(* CODESYS project Prepare.project

Project tree, tasks and I/O mapping:
  Device : CODESYS Control x86 Arca Control SM, 3S - Smart Software Solutions GmbH, version 3.5.8.0
    application Application
      libraries: Standard, * (System); Network, 3.5.7.0 (3S - Smart Software Solutions GmbH); Arca Motion Library, 1.0.4.14 (BonMET)
      task MainTask (cyclic, interval t#20ms, priority 1) calls Main
      hand blocks/
        function block AuxAxis_PowerOn [ST]
        data type Grab_Command
        function block Grab_Control [ST]
        function block Grab_Demo [ST]
        data type Grab_State
        function block Hand_Gesture [ST]
        data type Gesture_Type
        data type Error_Message
        function block Hand_Gesture_Demo [ST]
      program Main [ST]
      function block Organize_Hand_Command [ST]
      CNC Execute/
        function block CNC_Execute_Manager [ST]
      simple_functions/
        function block Value_Clamp [ST]
      TCPIP Control/
        data type Robot_Command_via_tcp
        data type Robot_State
        function block TCP_Command_Extract_And_Analysis [ST]
        function block TCPServerConnection [ST]
      Vision Control/
        function block Vision_Control [ST]
      global variables GVL
    SoftMotion General Axis Pool
*)

// Device/Application/hand blocks/Grab_Command
TYPE Grab_Command :
STRUCT
	Tip_Angle : REAL;
	Root_Angle : REAL;
	Clamp_Angle : REAL;
END_STRUCT
END_TYPE

// Device/Application/hand blocks/Grab_State
TYPE Grab_State :
STRUCT
	Tip_State : BOOL;
	Root_State : BOOL;
	Clamp_Angle : REAL;
END_STRUCT
END_TYPE

// Device/Application/hand blocks/Gesture_Type
{attribute 'qualified_only'}
{attribute 'strict'}
TYPE Gesture_Type :
(
	Gesture_Type_None			:= 0,
	Gesture_Type_Num_1		:= 1,
	Gesture_Type_Num_2		:= 2,
	Gesture_Type_Num_3		:= 3,
	Gesture_Type_Num_4		:= 4,
	Gesture_Type_Num_5		:= 5,
	Gesture_Type_Num_6		:= 6,
	Gesture_Type_Fist			:= 10,
	Gesture_Type_Palm			:= 11,
	Gesture_Type_ThumbUp		:= 12,
	Gesture_Type_ThumbDown	:= 13,
	Gesture_Type_ComeOnBaby	:= 14,
	Gesture_Type_PointTo		:= 15,
	Gesture_Type_Wave			:= 16,
	Gesture_Type_Nya			:= 17,
	Gesture_Type_MovObj			:= 18
);
END_TYPE

// Device/Application/hand blocks/Error_Message
{attribute 'qualified_only'}
{attribute 'strict'}
TYPE Error_Message :
(
	Err_None := 0,
	
	Err_AuxAxis_Movement_Cannot_read_virture_robot_position := 10,	// gesture block not reading robot position
	Err_Gesture_Type_Hand_Pos_Not_Given := 20,	// gesture block not given position
	Err_AuxAxis_Movement_Block_err := 30,	// gesture block first reset movement block err
	Err_Gesture_Type_Cycle_mov_block_err := 40,	// gesture block cycle movement block err
	
	Err_PowerOn_Block_Err := 50,
	Err_PowerOn_TimeOut := 51,
	
	Err_Power_Reset_Block_Err := 60,
	Err_Power_Reset_TimeOut := 61,
	
	Err_Group_Enable_Block_Err := 70,
	Err_Group_Enable_TimeOut := 71
);
END_TYPE

// Device/Application/TCPIP Control/Robot_Command_via_tcp
TYPE Robot_Command_via_tcp :
STRUCT
	X_Axis_Valid : BOOL;
	X_value : REAL;
	Y_Axis_Valid : BOOL;
	Y_value : REAL;
	Z_Axis_Valid : BOOL;
	Z_value : REAL;
	Spin : BOOL;
	Grab_Valid : BOOL;
	Grab_state : BOOL := FALSE;
	Gesture_Valid : BOOL;
	Gesture_Num : Gesture_Type;
	Enabl_Hand_Valid : BOOL;
	Enabl_Hand_state : BOOL;
	Gesture_Demo_Valid : BOOL;
	Gesture_Demo_state : BOOL;
	CNC_Mov_Valid : BOOL;
	CNC_Mov_Program_Num : INT;
END_STRUCT
END_TYPE

// Device/Application/TCPIP Control/Robot_State
TYPE Robot_State :
STRUCT
	Hand_Enabled : BOOL;
	Hand_Enb_Err : BOOL;
	Grab_State : BOOL;
	Gesture_State : Gesture_Type := gesture_type.Gesture_Type_None;
	Hand_Mov_Err : BOOL;
	Robot_Mov_Err : BOOL;
	CNC_Executing : BOOL;
	CNC_Execute_Done : BOOL;
	CNC_Execute_Err : BOOL;
END_STRUCT
END_TYPE

// Device/Application/GVL
VAR_GLOBAL
	AllAxisGroupEnb : BOOL := FALSE;
END_VAR

// Device/Application/Main
PROGRAM Main
VAR
	// manual function
	enable_internal : BOOL;
	MoveEn:BOOL:=FALSE;
	enb_triger : r_trig;
	disenb_triger : r_trig;
	
	start_hand_demo_internal : BOOL;
	demo_triger : r_trig;
	
	GestInternal: BOOL;
	GestTypeInternal:INT;
	Gest_triger : R_TRIG;
	
	// auto function
	TCP_Server : TCPserverconnection;
	commandOut : TCP_Command_Extract_And_Analysis;
	handMov : Organize_Hand_Command;
	Execute_CNC_Via_TCP : CNC_Execute_Manager;
	vision : vision_control;
	hand_cmd_valid : BOOL;
	hand_cmd : robot_command_via_tcp;
	old_pos_ready, new_pos_ready : BOOL;
	pick_triger, release_triger : R_TRIG;
	
	//debug
	ToqueT : ARRAY [0..13] OF ArcaLibrary.MCAT_AxisSetLimits;
	Texe : BOOL;
	Tdone, Terr : ARRAY [0..13] OF BOOL;
	SpL, TqL : ARRAY [1..13] OF REAL;
	ToqueState : INT := 0;
	axisOffset : INT := 13;
	axisMaxNum : INT := 25;
	i : INT;
	debug_auto_torque : BOOL;
	ToqueLimit: REAL := 0.5;
	
	AxisM : ARRAY [1..13] OF MCAT_ReadAxisMeasures;
	Aenb : BOOL := TRUE;
	Availd : ARRAY [1..13] OF BOOL;
	AtqM : ARRAY [1..13] OF REAL;
	
	tryRPow : ARRAY [1..13] OF ArcaLibrary.MCAT_ReadPowerStatus;
	PowS : ARRAY [1..13] OF byte;
	clk: INT;
	
	
	/// one button on
	EnableOld:BOOL:=FALSE;
	Status:INT;
	GoToZero:BOOL:=FALSE;
	CycleDone:BOOL;
	
	MoveAbsBlocks:ARRAY[0..5] OF ArcaLibrary.MC_MoveAbsolute;
	PosZero : ARRAY[0..5] OF REAL := [0.0,  18.0, 32.0, 0.0, 0.0, 0.0];
	ExecuteZero:BOOL:=FALSE;
	SpeedZero:REAL:=0.1;
	AccelZero:REAL:=5.0;
	DecelZero:REAL:=5.0;
	JerkZero:REAL:=50.0;
	ZeroError:BOOL;
	ZeroDone:BOOL;
	
	AxPos:ARRAY[1..12] OF REAL;
	AxPosRef:ARRAY[1..12] OF REAL;
	AxReadMea:ARRAY[1..12] OF ArcaLibrary.MCAT_ReadAxisMeasures;
	AxReadRef:ARRAY[1..12] OF ArcaLibrary.MCAT_ReadAxisRef;
	
	AxMoveAbs : ArcaLibrary.MC_MoveAbsolute;
	AxMoveAbs2 : ArcaLibrary.MC_MoveAbsolute;
	AxMoveEn:BOOL:=FALSE;
	AxMoveN:INT:=0;
	AxMovePos:REAL:=0;
	AxMoveVel:REAL:=1;
	AxMoveAcc:REAL:=1;
	AxMoveJerk:REAL:=25.0;
	AxMoveDone:BOOL;
	AxMoveDone2:BOOL;
	
	GrpEn:ArcaLibrary.MC_GroupEnable;
	GrpDis:ArcaLibrary.MC_GroupDisable;
	GrpEnDone, GrpEnErr:BOOL;
	GrpRead:ArcaLibrary.MC_GroupReadActualPosition;
	GrpPos:ARRAY[1..6] OF REAL;

	//initial position of the tool:
	Pos1 : ARRAY[0..5] OF REAL := [0.36, 0.000, 0.7, 0.000, 10, -180.000];
	Pos2 : ARRAY[0..5] OF REAL := [0.36, 0.010, 0.65, 0.000, 10, -180.000];
	Pos3 : ARRAY[0..5] OF REAL := [0.36, -0.010, 0.7, 0.000, 10, -180.000];
	Pos4 : ARRAY[0..5] OF REAL := [0.36, 0.000, 0.65, 0.000, 10, -180.000];
	
	Posleft : ARRAY[0..5] OF REAL := [-60.0,  7.0, 27.0, 0.0, 0.0, 0.0];
	Posright : ARRAY[0..5] OF REAL := [-50.0,  9.0, 30.0, 0.0, 0.0, 0.0];
	
	
	ToolMoveAbs1, ToolMoveAbs2, ToolMoveAbs3, ToolMoveAbs4, ToolMoveAbs5, ToolMoveAbs6 : ArcaLibrary.MC_MoveLinearAbsolute;
	ToolMoveDone1, ToolMoveDone2, ToolMoveDone3, ToolMoveDone4, ToolMoveDone5, ToolMoveDone6 :BOOL;
	
	ToolMoveVel:REAL:=1;
	ToolMoveAcc:REAL:=100;
	ToolMoveJrk:REAL:=1000;
	
	BlendMov : ArcaLibrary.MC_BUFFER_MODE := mcBuffered;
	TransMov : ArcaLibrary.MC_TRANSITION_MODE := tmCornerDistance;	
	TransPar : REAL := 0.0;
	
	ReadDI: ArcaLibrary.BMET_Read_DI;
	ReadDO: ArcaLibrary.BMET_Read_DO;
	WriteDO: ArcaLibrary.BMET_Write_DO;
	ValueRead : UINT;
	ValueDO : UINT;
	LampActivate : UINT;
	
	J : INT := 0;
	DelayTimer : Ton;
END_VAR

//	manually operation process
enb_triger (clk := enable_internal);
disenb_triger (clk := NOT enable_internal);
demo_triger (clk := start_hand_demo_internal);
Gest_triger (clk := GestInternal);

//*****************
TCP_Server(enable := TRUE, outDataReady := commandout.Response_Valid,
	 OutData := commandout.Response ,outDataSize := commandout.Response_Data_Size);

commandout(indata := tcp_server.InData 
	, inDataSize := TCP_Server.InDataSize
	, inData_Valid := TCP_Server.InDataReady
	, OutRobot_State := handmov.Current_Hand_State
	);
	
hand_cmd_valid := commandout.Command_Valid OR pick_triger.Q OR release_triger.Q OR enb_triger.Q
	OR disenb_triger.Q OR demo_triger.Q
	OR Gest_triger.Q;
hand_cmd := commandout.Command;
IF pick_triger.Q THEN
	hand_cmd.Gesture_Valid := TRUE;
	hand_cmd.Gesture_Num := 10;
END_IF
IF release_triger.Q THEN
	hand_cmd.Gesture_Valid := TRUE;
	hand_cmd.Gesture_Num := 11;
END_IF
IF enb_triger.Q THEN
	hand_cmd.Enabl_Hand_Valid := TRUE;
	hand_cmd.Enabl_Hand_state := TRUE;
END_IF
IF disenb_triger.Q THEN
	hand_cmd.Enabl_Hand_Valid := TRUE;
	hand_cmd.Enabl_Hand_state := FALSE;
END_IF
IF demo_triger.Q THEN
	hand_cmd.Gesture_Demo_Valid := TRUE;
	hand_cmd.Gesture_Demo_state := TRUE;
END_IF
IF Gest_triger.Q THEN
	hand_cmd.Gesture_Valid := TRUE;
	hand_cmd.Gesture_Num := GestTypeInternal;
END_IF

handMov(enable:= TRUE, new_cmd_valid := hand_cmd_valid
	, new_cmd := hand_cmd
	);

Execute_CNC_Via_TCP(enable := TRUE, mov_group := 1
	, Tcp_cmd_valid := commandout.Command_Valid
	, TCP_CMD := commandout.Command
	);
(*	dont where has conflict, after enable second robot keep sotping cannot move
vision(enable := handmov.Current_Hand_State.Hand_Enabled, robot_group := 1
	, execute := vision.ready
	, wait_signal_before_pick := TRUE, isPicked := handmov.Current_Hand_State.Gesture_State = 10
	, delay_release_obj := T#2S
	);

pick_triger(clk := vision.ready_to_pick);
release_triger(clk := vision.ready_to_release);
*)
(*************************
	Toque test above
**************************)
ToqueT[01](Execute := Texe, Axis := 06, SpeedLimit := SpL[01], TorqueLimit := TqL[01], Done => Tdone[01], Error => Terr [01]);
ToqueT[02](Execute := Texe, Axis := 07, SpeedLimit := SpL[02], TorqueLimit := TqL[02], Done => Tdone[02], Error => Terr [02]);
ToqueT[03](Execute := Texe, Axis := 08, SpeedLimit := SpL[03], TorqueLimit := TqL[03], Done => Tdone[03], Error => Terr [03]);
ToqueT[04](Execute := Texe, Axis := 09, SpeedLimit := SpL[04], TorqueLimit := TqL[04], Done => Tdone[04], Error => Terr [04]);
ToqueT[05](Execute := Texe, Axis := 10, SpeedLimit := SpL[05], TorqueLimit := TqL[05], Done => Tdone[05], Error => Terr [05]);
ToqueT[06](Execute := Texe, Axis := 11, SpeedLimit := SpL[06], TorqueLimit := TqL[06], Done => Tdone[06], Error => Terr [06]);
ToqueT[07](Execute := Texe, Axis := 12, SpeedLimit := SpL[07], TorqueLimit := TqL[07], Done => Tdone[07], Error => Terr [07]);
ToqueT[08](Execute := Texe, Axis := 13, SpeedLimit := SpL[08], TorqueLimit := TqL[08], Done => Tdone[08], Error => Terr [08]);
ToqueT[09](Execute := Texe, Axis := 14, SpeedLimit := SpL[09], TorqueLimit := TqL[09], Done => Tdone[09], Error => Terr [09]);
ToqueT[10](Execute := Texe, Axis := 15, SpeedLimit := SpL[10], TorqueLimit := TqL[10], Done => Tdone[10], Error => Terr [10]);
ToqueT[11](Execute := Texe, Axis := 16, SpeedLimit := SpL[11], TorqueLimit := TqL[11], Done => Tdone[11], Error => Terr [11]);

// auto set toque limit after axis enabled
CASE ToqueState OF 
	0:
		IF handMov.Current_Hand_State.Hand_Enabled AND NOT debug_auto_torque THEN
			i := 0;
			toquestate := 10;
		END_IF
	10:
		ToqueT[i](Execute := TRUE, Axis := axisOffset + i, TorqueLimit := ToqueLimit, Done => Tdone[i], Error => Terr [i]);
		IF Tdone[i] THEN
			i := i + 1;
			IF axisOffset + i > axisMaxNum THEN
				i := 0;
				toquestate := 20;
			END_IF
		END_IF
	20:
		ToqueT[i](Execute := FALSE);
		i := i + 1;
		IF axisOffset + i > axisMaxNum THEN
			toquestate := 30;
		END_IF
	30:
		IF NOT handMov.Current_Hand_State.Hand_Enabled THEN
			toquestate := 0;
		END_IF
END_CASE

AxisM[01](enable := Aenb, Axis := 6, Torque=> AtqM[01]);
AxisM[02](enable := Aenb, Axis := 7, Torque=> AtqM[02]);
AxisM[03](enable := Aenb, Axis := 8, Torque=> AtqM[03]);
AxisM[04](enable := Aenb, Axis := 9, Torque=> AtqM[04]);
AxisM[05](enable := Aenb, Axis := 10, Torque=> AtqM[05]);
AxisM[06](enable := Aenb, Axis := 11, Torque=> AtqM[06]);
AxisM[07](enable := Aenb, Axis := 12, Torque=> AtqM[07]);
AxisM[08](enable := Aenb, Axis := 13, Torque=> AtqM[08]);
AxisM[09](enable := Aenb, Axis := 14, Torque=> AtqM[09]);
AxisM[10](enable := Aenb, Axis := 15, Torque=> AtqM[10]);
AxisM[11](enable := Aenb, Axis := 16, Torque=> AtqM[11]);

tryRPow[01](enable := TRUE, axis := 06, state=> pows[01]);
tryRPow[02](enable := TRUE, axis := 07, state=> pows[01]);
tryRPow[03](enable := TRUE, axis := 08, state=> pows[01]);
tryRPow[04](enable := TRUE, axis := 09, state=> pows[01]);
tryRPow[05](enable := TRUE, axis := 10, state=> pows[01]);
tryRPow[06](enable := TRUE, axis := 11, state=> pows[01]);
tryRPow[07](enable := TRUE, axis := 12, state=> pows[01]);
tryRPow[08](enable := TRUE, axis := 13, state=> pows[01]);
tryRPow[09](enable := TRUE, axis := 14, state=> pows[01]);
tryRPow[10](enable := TRUE, axis := 15, state=> pows[01]);
tryRPow[11](enable := TRUE, axis := 16, state=> pows[01]);


(***********************
one button start mov
************************)
// read of  measures
AxReadMea[1](Axis:=0, Enable:=(Status>=3 AND Status<100), Pos=>AxPos[1]);
AxReadMea[2](Axis:=1, Enable:=(Status>=3 AND Status<100), Pos=>AxPos[2]);
AxReadMea[3](Axis:=2, Enable:=(Status>=3 AND Status<100), Pos=>AxPos[3]);
AxReadMea[4](Axis:=3, Enable:=(Status>=3 AND Status<100), Pos=>AxPos[4]);
AxReadMea[5](Axis:=4, Enable:=(Status>=3 AND Status<100), Pos=>AxPos[5]);
AxReadMea[6](Axis:=5, Enable:=(Status>=3 AND Status<100), Pos=>AxPos[6]);
AxReadMea[7](Axis:=6, Enable:=(Status>=3 AND Status<100), Pos=>AxPos[7]);
AxReadMea[8](Axis:=7, Enable:=(Status>=3 AND Status<100), Pos=>AxPos[8]);
AxReadMea[9](Axis:=8, Enable:=(Status>=3 AND Status<100), Pos=>AxPos[9]);
AxReadMea[10](Axis:=9, Enable:=(Status>=3 AND Status<100), Pos=>AxPos[10]);
AxReadMea[11](Axis:=10, Enable:=(Status>=3 AND Status<100), Pos=>AxPos[11]);
AxReadMea[12](Axis:=11, Enable:=(Status>=3 AND Status<100), Pos=>AxPos[12]);
// read of reference
AxReadRef[1](Axis:=0, Enable:=(Status>=3 AND Status<100), PosRef=>AxPosRef[1]);
AxReadRef[2](Axis:=1, Enable:=(Status>=3 AND Status<100), PosRef=>AxPosRef[2]);
AxReadRef[3](Axis:=2, Enable:=(Status>=3 AND Status<100), PosRef=>AxPosRef[3]);
AxReadRef[4](Axis:=3, Enable:=(Status>=3 AND Status<100), PosRef=>AxPosRef[4]);
AxReadRef[5](Axis:=4, Enable:=(Status>=3 AND Status<100), PosRef=>AxPosRef[5]);
AxReadRef[6](Axis:=5, Enable:=(Status>=3 AND Status<100), PosRef=>AxPosRef[6]);
AxReadRef[7](Axis:=6, Enable:=(Status>=3 AND Status<100), PosRef=>AxPosRef[7]);
AxReadRef[8](Axis:=7, Enable:=(Status>=3 AND Status<100), PosRef=>AxPosRef[8]);
AxReadRef[9](Axis:=8, Enable:=(Status>=3 AND Status<100), PosRef=>AxPosRef[9]);
AxReadRef[10](Axis:=9, Enable:=(Status>=3 AND Status<100), PosRef=>AxPosRef[10]);
AxReadRef[11](Axis:=10, Enable:=(Status>=3 AND Status<100), PosRef=>AxPosRef[11]);
AxReadRef[12](Axis:=11, Enable:=(Status>=3 AND Status<100), PosRef=>AxPosRef[12]);
// read group position MCS
GrpRead(AxesGroup:=0, Execute:=(Status>=3 AND Status<100), 
	CoordSystem:=ArcaLibrary.MC_COORD_SYSTEM.mcMcs, Position=>GrpPos);

// Powered acquisition from panel 读轴的输入输出
ReadDI(Axis:=0,Enable:=TRUE,Value=>ValueRead);
ReadDO(Axis:=0,Enable:=TRUE,Value=>ValueDO);
WriteDO(Axis:=0,Enable:=TRUE,Value:=0, Mask:=15);


//Press EnableServo to turn on the motors
IF (ValueRead=8) THEN
	J := J + 1;
	IF (J>50) THEN
		enable_internal:=TRUE;
	END_IF
END_IF
//if Button EnableServo is pressed for more than 1 second, turn off the motors
IF (ValueRead=8 AND J > 150) THEN  //OR (ValueRead=0) THEN
	enable_internal:=FALSE;
	MoveEn:=FALSE;
	J:=0;
END_IF

//
// State machines
//
IF (NOT enable_internal) THEN
	WriteDO(Axis:=0,Enable:=TRUE,Value:=0,Mask:=15);
	Status:=0;
ELSE
	WriteDO(Axis:=0,Enable:=TRUE,Value:=2,Mask:=15);
END_IF

//ReadDigitalInput as MoveEnable
IF (ValueRead=16) THEN
	MoveEn:=TRUE;
END_IF
IF (ValueRead=32) THEN
	MoveEn:=FALSE;
END_IF

CASE (Status) OF
	
	//// OFF
	0:
	IF (enable_internal) THEN
		WriteDO(Axis:=0,Enable:=TRUE,Value:=2,Mask:=15);
		Status:=1;
	END_IF
	
	//// POWERING ON
	1:
		IF AllAxisGroupEnb THEN
			Status:=2;
		END_IF
	
	//// IDLE - WAIT FOR COMMAND
	2:
		IF moveEn THEN
			AxMoveAbs(Axis:=11, execute := FALSE);
			status := 3;
		END_IF
	// FORWARD KINEMATIC
	3:
		WriteDO(Axis:=0,Enable:=TRUE,Value:=3,Mask:=15);
		IF NOT moveEn THEN
			status := 2;
		END_IF
			
		// move 5axis of robot 1, in order to move robot later
		AxMoveAbs(Axis:=11, Execute:=TRUE, Position:=80, Velocity:=10, 
			Acceleration:=10, Deceleration:=10, Jerk:=10, 
			BufferMode:=ArcaLibrary.MC_BUFFER_MODE.mcAborting, Done=>AxMoveDone);
					
		IF AxMoveDone THEN
			AxMoveAbs(Axis:=11, execute := FALSE);
			status := 4;
		END_IF
	
	// GROUP MOVEMENT - START
	4:
		WriteDO(Axis:=0,Enable:=TRUE,Value:=6,Mask:=15);
		IF (NOT MoveEn) THEN
			WriteDO(Axis:=0,Enable:=TRUE,Value:=3,Mask:=15);
			Status:=3;
		END_IF
		
		CycleDone:=FALSE;
		// clear block status
		ToolMoveAbs1(AxesGroup:=1, Execute:=FALSE);
		ToolMoveAbs2(AxesGroup:=1, Execute:=FALSE);
		ToolMoveAbs3(AxesGroup:=1, Execute:=FALSE);
		ToolMoveAbs4(AxesGroup:=1, Execute:=FALSE);
		ToolMoveAbs5(AxesGroup:=1, Execute:=FALSE);
		ToolMoveAbs6(AxesGroup:=1, Execute:=FALSE);
		Status:=5;
		DelayTimer(in:= FALSE);
		CycleDone:=FALSE;
		GestInternal := FALSE;
		
			
	// GROUP MOVEMENT - FIRST MOVEMENT
	5:
		WriteDO(Axis:=0,Enable:=TRUE,Value:=6,Mask:=15);
		IF (NOT MoveEn) THEN
			Status:=3;
		END_IF
		
		IF (NOT CycleDone) THEN
			ToolMoveAbs1(AxesGroup:=1, Execute:=TRUE, Position:=ADR(Pos1), Velocity:=ToolMoveVel, Acceleration:=ToolMoveAcc,
				Deceleration:=ToolMoveAcc, Jerk:=ToolMoveJrk, CoordSystem:=mcMcs 
				, TransitionMode := tmNone
				, BufferMode:=mcBuffered, Done=>ToolMoveDone1);
		END_IF
		
		IF (ToolMoveDone1) THEN
			GestInternal := TRUE;
			GestTypeInternal := 1;
			DelayTimer(in:= TRUE, pt := T#5000MS);
			IF delaytimer.Q THEN
				DelayTimer(in:= FALSE);
				GestInternal := FALSE;
				Status:= 51;
				ToolMoveDone1 := FALSE;
			END_IF
		END_IF
	
		
	// GROUP MOVEMENT - SECOND MOVEMENT
	51:
		WriteDO(Axis:=0,Enable:=TRUE,Value:=6,Mask:=15);
		IF (NOT MoveEn) THEN
			Status:=3;
		END_IF
		
		IF (NOT CycleDone) THEN
			ToolMoveAbs2(AxesGroup:=1, Execute:=TRUE, Position:=ADR(Pos2), Velocity:=ToolMoveVel, Acceleration:=ToolMoveAcc,
				Deceleration:=ToolMoveAcc, Jerk:=ToolMoveJrk, CoordSystem:=ArcaLibrary.MC_COORD_SYSTEM.mcMcs, 
				BufferMode:=BlendMov, TransitionMode:=TransMov, TransitionParameter:=ADR(TransPar), Done=>ToolMoveDone2);
		END_IF
		
		IF (ToolMoveDone2) THEN
			GestInternal := TRUE;
			GestTypeInternal := 2;
			DelayTimer(in:= TRUE, pt := T#5000MS);
			IF delaytimer.Q THEN
				DelayTimer(in:= FALSE);
				GestInternal := FALSE;
				Status:=52;
			END_IF
		END_IF

	// GROUP MOVEMENT - THIRD MOVEMENT
	52:
		WriteDO(Axis:=0,Enable:=TRUE,Value:=6,Mask:=15);
		IF (NOT MoveEn) THEN
			Status:=3;
		END_IF
		
		IF (NOT CycleDone) THEN
			ToolMoveAbs3(AxesGroup:=1, Execute:=TRUE, Position:=ADR(Pos3), Velocity:=ToolMoveVel, Acceleration:=ToolMoveAcc,
				Deceleration:=ToolMoveAcc, Jerk:=ToolMoveJrk, CoordSystem:=ArcaLibrary.MC_COORD_SYSTEM.mcMcs, 
				BufferMode:=BlendMov, TransitionMode:=TransMov, TransitionParameter:=ADR(TransPar), Done=>ToolMoveDone3);
		END_IF
		
		IF (ToolMoveDone3) THEN
			GestInternal := TRUE;
			GestTypeInternal := 3;
			DelayTimer(in:= TRUE, pt := T#5000MS);
			IF delaytimer.Q THEN
				DelayTimer(in:= FALSE);
				GestInternal := FALSE;
				Status:=4;
			END_IF
		END_IF

	// GROUP MOVEMENT - FOURTH MOVEMENT
	53:
		WriteDO(Axis:=0,Enable:=TRUE,Value:=6,Mask:=15);
		IF (NOT MoveEn) THEN
			Status:=3;
		END_IF
		
		IF (NOT CycleDone) THEN
			ToolMoveAbs4(AxesGroup:=1, Execute:=TRUE, Position:=ADR(Pos4), Velocity:=ToolMoveVel, Acceleration:=ToolMoveAcc,
				Deceleration:=ToolMoveAcc, Jerk:=ToolMoveJrk, CoordSystem:=ArcaLibrary.MC_COORD_SYSTEM.mcMcs, 
				BufferMode:=mcBuffered, Done=>ToolMoveDone4);
		END_IF

		IF (ToolMoveDone4) THEN
			Status:=4;
		END_IF

	// GROUP MOVEMENT - FIFTH MOVEMENT
	54:
		WriteDO(Axis:=0,Enable:=TRUE,Value:=6,Mask:=15);
		IF (NOT MoveEn) THEN
			Status:=3;
		END_IF
		
		IF (NOT CycleDone) THEN
	//		ToolMoveAbs5(AxesGroup:=1, Execute:=TRUE, Position:=ADR(Pos4), Velocity:=ToolMoveVel, Acceleration:=ToolMoveAcc,
	//			Deceleration:=ToolMoveAcc, Jerk:=ToolMoveJrk, CoordSystem:=ArcaLibrary.MC_COORD_SYSTEM.mcMcs, 
	//			BufferMode:=BlendMov, TransitionMode:=TransMov, TransitionParameter:=ADR(TransPar), Done=>ToolMoveDone5);
		END_IF

		IF (ToolMoveDone5) THEN
			Status:=55;
		END_IF

	// GROUP MOVEMENT - SIXTH MOVEMENT
	55:
		WriteDO(Axis:=0,Enable:=TRUE,Value:=6,Mask:=15);
		IF (NOT MoveEn) THEN
			Status:=3;
		END_IF
		
		IF (NOT CycleDone) THEN
	//		ToolMoveAbs6(AxesGroup:=1, Execute:=TRUE, Position:=ADR(Pos3), Velocity:=ToolMoveVel, Acceleration:=ToolMoveAcc,
	//			Deceleration:=ToolMoveAcc, Jerk:=ToolMoveJrk, CoordSystem:=ArcaLibrary.MC_COORD_SYSTEM.mcMcs, 
	//			BufferMode:=BlendMov, TransitionMode:=TransMov, TransitionParameter:=ADR(TransPar), Done=>ToolMoveDone6);
		END_IF

		IF (ToolMoveDone6) THEN
			CycleDone:=TRUE;
			Status:=4;
		END_IF


	//// ERROR
	100:
		WriteDO(Axis:=0,Enable:=TRUE,Value:=3,Mask:=15);
	
	
END_CASE

END_PROGRAM

// Device/Application/TCPIP Control/TCPServerConnection
FUNCTION_BLOCK TCPServerConnection
VAR_INPUT
	Enable : BOOL;
	OutDataReady : BOOL;
	OutDataSize : CAA.SIZE;
	OutData :  ARRAY [0..255] OF BYTE;;
END_VAR
VAR_OUTPUT
	Err : BOOL;
	InDataReady : BOOL;
	InDataSize : CAA.SIZE;
	InData : STRING;
END_VAR
VAR
	TCPServer : NBS.TCP_Server;
	IP_Addr : NBS.IP_ADDR := (sAddr :='192.168.80.240');
	Port: UINT := 23; // TCP/IP port
	TCPS_Err : BOOL := FALSE;
	TCPS_Err_Mssage : NBS.ERROR;
	
	TCPS_Connection : NBS.TCP_Connection;
	
	ServerRead : NBS.TCP_Read;
	ServerSend : NBS.TCP_Write;
	
	Hendle_enable :BOOL;
	Some_Connect_In : BOOL;
	
	// message out
	_OutDataSize : CAA.SIZE;
	debug : BOOL;
	testTXT :STRING := '0123456';
	testByte : ARRAY [0..5] OF BYTE := [40,12,41,40,10,41];
	ddone, deErr, dxErr : BOOL;
END_VAR

// initialize TCP server
TCPServer(xEnable := Enable, ipAddr := IP_Addr, uiPort := Port, xError => TCPS_Err, eError => TCPS_Err_Mssage);

// send handle after there are some client connect 
TCPS_Connection(xEnable := Hendle_enable, hServer := TCPServer.hServer);

// enable handle after tcp server is online, up below command is insure if there is a client disconnect, the command will be turn off one cycle
IF TCPServer.xBusy AND NOT Hendle_enable THEN
	Hendle_enable := TRUE;
ELSIF NOT TCPServer.xBusy AND Hendle_enable THEN
	Hendle_enable := FALSE;
END_IF

// some one connect in
IF TCPS_Connection.xActive THEN
	Some_Connect_In := TRUE;
END_IF

// health check, if connection broken then turn off handle to wait next connection
IF Some_Connect_In AND NOT TCPS_Connection.xActive THEN
	Some_Connect_In := Hendle_enable := FALSE;
END_IF

// receive data from client
ServerRead(xEnable := TCPS_Connection.xActive, hConnection := TCPS_Connection.hConnection
	, szSize := SIZEOF(InData)
	, pData := ADR(InData)
	, szCount => InDataSize
	, xReady => InDataReady	// when new data comes this flag will be true in one cycle
	);

	
// send data to client
IF OutDataSize > 0 THEN
	_OutDataSize := OutDataSize;
ELSE
	_OutDataSize := SIZEOF(OutData);
END_IF

IF outdataReady THEN
	debug := TRUE;
END_IF

ServerSend(xExecute := OutDataReady, hConnection := TCPS_Connection.hConnection, szSize := _OutDataSize, pData := ADR(OutData), udiTimeOut := 1000
	, xError => dxErr, xDone => ddone);

END_FUNCTION_BLOCK

// Device/Application/TCPIP Control/TCP_Command_Extract_And_Analysis
FUNCTION_BLOCK TCP_Command_Extract_And_Analysis
VAR_INPUT
	InData : STRING;
	InDataSize : CAA.SIZE;
	InData_Valid : BOOL;
	OutRobot_State : Robot_State;
END_VAR
VAR_OUTPUT
	Command_Valid : BOOL;
	Command : robot_command_via_tcp;
	Response : ARRAY [0..255] OF BYTE;
	Response_Data_Size : CAA.SIZE;
	Response_Valid : BOOL;
	Error : BOOL;
	ErrorMassage : STRING;
END_VAR
VAR
	newDataSize : INT;
	i : INT;
	y : INT;
	state : INT := 0;
	charInData : POINTER TO BYTE;
	charStartF : BYTE := 40; // (
	charStartS : BYTE := 41; // )
	charMid : BYTE := 59; // ;
	charEndF : BYTE := 91; // [
	charEndS : BYTE := 93; // ]
	charAU : BYTE := 65;	// A
	charZU : BYTE := 90;	// Z
	charAL : BYTE := 97;	// a
	charZL : BYTE := 122;	// z
	charMinus : BYTE := 45; // -
	charPeriod : BYTE := 46; // .
	char0 : BYTE := 48; // 0
	char9 : BYTE := 57; // 9
	cache : ARRAY [0..10] OF BYTE;
	cacheCleaner : ARRAY [0..10] OF BYTE;
	
	tag : STRING;
	tagPointer : POINTER TO STRING;
	tagPass : STRING(12);
	
	content : STRING;
	contentPointer : POINTER TO STRING;
	contentNum : REAL;
	_defult_cmd : robot_command_via_tcp;
	
	
	// out going data process
	old_robot_state : Robot_State;
	old_gesture_state : ARRAY [0..8] OF BYTE := [40, 71, 101, 115, 116, 41, 48, 48, 59]; //(Gest)00;
	old_Grab_state : ARRAY [0..7] OF BYTE := [40, 71, 114, 97, 98, 41, 48, 59]; //(Grab)0;
	old_Hand_Enb_state : ARRAY [0..7] OF BYTE := [40, 72, 69, 110, 98, 41, 48, 59]; //(HEnb)0;
	old_Hand_Enb_Err_state : ARRAY [0..10] OF BYTE := [40, 72, 69, 110, 98, 69, 114, 114, 41, 48, 59]; //(HEnbErr)0;
	old_Hand_Mov_Err_state : ARRAY [0..10] OF BYTE := [40, 72, 77, 111, 118, 69, 114, 114, 41, 48, 59]; //(HMovErr)0;
	old_Robot_Mov_Err_state : ARRAY [0..10] OF BYTE := [40, 82, 77, 111, 118, 69, 114, 114, 41, 48, 59]; //(RMovErr)0;
	old_CNC_Executing_state : ARRAY [0..9] OF BYTE := [40, 67, 78, 67, 105, 110, 103, 41, 48, 59]; //(CNCing)0;
	old_CNC_Err_state : ARRAY [0..9] OF BYTE := [40, 67, 78, 67, 69, 72, 72, 41, 48, 59]; //(CNCErr)0;
	old_CNC_Done_state : ARRAY [0..10] OF BYTE := [40, 67, 78, 67, 68, 111, 110, 110, 41, 48, 59]; //(CNCDone)0;
	
	data_end : ARRAY [0..1] OF BYTE := [13, 10];
	og_i : INT;
	og_num_counter : INT;
	
	abc : INT;
	message_sending_timer : ton;
END_VAR

IF Command_Valid THEN
	command_Valid := FALSE; // reset flag after one cycle
	Command := _defult_cmd;	// all content value will only save for one cycle
END_IF;

// process income data
IF (INData_valid AND InDataSize > 0) THEN
	charInData := ADR(InData);
	newDataSize := UDINT_TO_INT(InDataSize);
	Error := FALSE;
	i := 0;
	WHILE i < newDataSize DO
		CASE state OF
			-9:
				IF charInData^ = 93 THEN
					Command_Valid := TRUE;
					i := i + 1;
					state := 0; // if read ]
				ELSE state := 999;
				END_IF
			-8:
				IF charInData^ = 10 THEN
					charInData := charInData + 1;
					i := i + 1;
					state := -9; // if read LF
				ELSE state := 999;
				END_IF
			-7:
				IF charInData^ = 91 THEN
					charInData := charInData + 1;
					i := i + 1;
					state := -8; // if read [
				ELSE state := 999;
				END_IF
			-6:
				IF charInData^ = 93 THEN
					charInData := charInData + 1;
					i := i + 1;
					state := -7; // if read ]
				ELSE state := 999;
				END_IF
			-5:
				IF charInData^ = 13 THEN
					charInData := charInData + 1;
					i := i + 1;
					state := -6; // if read CR
				ELSE state := 999;
				END_IF
			0:
				IF (charInData^ = charStartF) THEN // if read (
					charInData := charInData + 1;
					i := i + 1;
					y := 0;
					state := 10;
				ELSIF charInData^ = charEndF THEN // if read [
					charInData := charInData + 1;
					i := i + 1;
					state := -5;
				ELSE state := 999;
				END_IF
			10:	// exturct laybel
				// if is not ) and not reach end of text and no error
				WHILE (charInData^ <> charStartS) AND (i < newDataSize) AND state = 10 DO
					// if is reading english letter
					IF (CharInData^ >= charAU AND CharInData^ <= charZU) OR (CharInData^ >= charAL AND CharInData^ <= charZL) THEN	
						cache[y] := CharInData^;
						y := y + 1;
						i := i + 1;
						IF i < newDataSize THEN	// only move pointer futher if is not reach the end of text
							charInData := charInData + 1;
						END_IF
					ELSE state := 999;
					END_IF
				END_WHILE
				IF charInData^ = charStartS AND i < newDataSize THEN	// if is ) and not reach end of text
					charInData := charInData + 1;
					i := i + 1;
					y := 0;
					tagPointer := ADR(cache);
					tag := tagPointer^;
					cache := cacheCleaner;
					state := 20;
				END_IF
			20:	// extruct data
				// if is not ; and not reach end of text and no error
				WHILE (charInData^ <> charMid) AND (i < newDataSize) AND state = 20 DO
					// if is reading numbers and - and .
					IF (CharInData^ >= charMinus AND CharInData^ <= charPeriod) OR (CharInData^ >= char0 AND CharInData^ <= char9) THEN
						cache[y] := CharInData^;
						y := y + 1;
						i := i + 1;
						IF i < newDataSize THEN	// only move pointer futher if is not reach the end of text
							charInData := charInData + 1;
						END_IF
					ELSE state := 999;
					END_IF
				END_WHILE
				IF charInData^ = charMid AND i < newDataSize THEN	// if is ; and not reach end of text
					charInData := charInData + 1;
					i := i + 1;
					y := 0;
					contentPointer := ADR(cache);
					content := contentPointer^;
					cache := cacheCleaner;
					contentNum := STRING_TO_REAL(content);
					state := 30;
				END_IF
			30:	// asign data, new label add here
				IF tag = 'X' THEN
					Command.X_Axis_Valid := TRUE;
					Command.X_value := contentNum;
				ELSIF tag = 'Y' THEN
					Command.Y_Axis_Valid := TRUE;
					Command.Y_value := contentNum;
				ELSIF tag = 'Z' THEN
					Command.Z_Axis_Valid := TRUE;
					Command.Z_value := contentNum;
				ELSIF tag = 'GRAB' THEN
					Command.Grab_Valid := TRUE;
					IF contentNum = 1 THEN
						Command.Grab_state := TRUE;
					ELSE 
						Command.Grab_state := FALSE;
					END_IF
				ELSIF tag = 'GEST' THEN
					Command.Gesture_Valid := TRUE;
					CASE (REAL_TO_INT(contentnum)) OF
						0:
							Command.Gesture_Num := 0;
						1:
							Command.Gesture_Num := 1;
						2:
							Command.Gesture_Num := 2;
						3:
							Command.Gesture_Num := 3;
						4:
							Command.Gesture_Num := 4;
						5:
							Command.Gesture_Num := 5;
						6:
							Command.Gesture_Num := 6;
						10:
							Command.Gesture_Num := 10;
						11:
							Command.Gesture_Num := 11;
						12:
							Command.Gesture_Num := 12;
						13:
							Command.Gesture_Num := 13;
						14:
							Command.Gesture_Num := 14;
						15:
							Command.Gesture_Num := 15;
						16:
							Command.Gesture_Num := 16;
						17:
							Command.Gesture_Num := 17;
					END_CASE
					
				ELSIF tag = 'HENB' THEN	// hand enable
					Command.Enabl_Hand_Valid := TRUE;
					IF contentNum = 1 THEN
						Command.Enabl_Hand_state := TRUE;
					ELSE 
						Command.Enabl_Hand_state := FALSE;
					END_IF
				ELSIF tag = 'HDem' THEN	// hand demo
					Command.Gesture_Demo_Valid := TRUE;
					IF contentNum = 1 THEN
						Command.Gesture_Demo_state := TRUE;
					ELSE 
						Command.Gesture_Demo_state := FALSE;
					END_IF
				ELSIF tag = 'CNC' THEN	// CNC program move command
					Command.CNC_Mov_Valid := TRUE;
					Command.CNC_Mov_Program_Num := REAL_TO_INT(contentnum);
				END_IF
				state := 0;
			999:
				i := newDataSize;
				state := 0;
				Error := TRUE;
				ErrorMassage := 'Error Data not match rule';
		END_CASE
	END_WHILE
END_IF

Response_Valid := FALSE;
message_sending_timer(in := TRUE, pt := T#100MS);
// process outgoing data
IF
	(
	outrobot_state.Gesture_State <> old_robot_state.Gesture_State
	OR outrobot_state.Grab_State <> old_robot_state.Grab_State
	OR outrobot_state.Hand_Enabled <> old_robot_state.Hand_Enabled
	OR outrobot_state.Hand_Enb_Err <> old_robot_state.Hand_Enb_Err
	OR outrobot_state.Hand_Mov_Err <> old_robot_state.Hand_Mov_Err
	OR outrobot_state.Robot_Mov_Err <> old_robot_state.Robot_Mov_Err
	)
	AND
	message_sending_timer.Q
THEN
	message_sending_timer(in := FALSE);
	abc := abc +1;
	//debug:= TRUE;
	og_num_counter := 0;
	
	// gesture state
	IF outrobot_state.Gesture_State <> old_robot_state.Gesture_State THEN
			
		CASE outrobot_state.Gesture_State OF
			0:
				old_gesture_state[6] := 48;
				old_gesture_state[7] := 48;
			1:
				old_gesture_state[6] := 48;
				old_gesture_state[7] := 49;
			2:
				old_gesture_state[6] := 48;
				old_gesture_state[7] := 50;
			3:
				old_gesture_state[6] := 48;
				old_gesture_state[7] := 51;
			4:
				old_gesture_state[6] := 48;
				old_gesture_state[7] := 52;
			5:
				old_gesture_state[6] := 48;
				old_gesture_state[7] := 53;
			6:
				old_gesture_state[6] := 48;
				old_gesture_state[7] := 54;
			10:
				old_gesture_state[6] := 49;
				old_gesture_state[7] := 48;
			11:
				old_gesture_state[6] := 49;
				old_gesture_state[7] := 49;
			12:
				old_gesture_state[6] := 49;
				old_gesture_state[7] := 50;
			13:
				old_gesture_state[6] := 49;
				old_gesture_state[7] := 51;
			14:
				old_gesture_state[6] := 49;
				old_gesture_state[7] := 52;
			15:
				old_gesture_state[6] := 49;
				old_gesture_state[7] := 53;
			16:
				old_gesture_state[6] := 49;
				old_gesture_state[7] := 54;
			17:
				old_gesture_state[6] := 49;
				old_gesture_state[7] := 55;
		END_CASE
		
		FOR og_i := 0 TO UDINT_TO_INT(SIZEOF(old_gesture_state)) - 1 DO
			Response[og_num_counter] := old_gesture_state[og_i];
			og_num_counter := og_num_counter + 1;
		END_FOR
	END_IF
	
	// Grab state
	IF outrobot_state.Grab_State <> old_robot_state.Grab_State THEN
		IF outrobot_state.Grab_State THEN	// if true
			old_Grab_state[6] := 49;
		ELSE
			old_Grab_state[6] := 48;
		END_IF
		
		FOR og_i := 0 TO UDINT_TO_INT(SIZEOF(old_Grab_state)) - 1 DO
			Response[og_num_counter] := old_Grab_state[og_i];
			og_num_counter := og_num_counter + 1;
		END_FOR
	END_IF
	
	// hand enable state
	IF outrobot_state.Hand_Enabled <> old_robot_state.Hand_Enabled THEN
		IF outrobot_state.Hand_Enabled THEN	// if true
			old_Hand_Enb_state[6] := 49;
		ELSE
			old_Hand_Enb_state[6] := 48;
		END_IF
		
		FOR og_i := 0 TO UDINT_TO_INT(SIZEOF(old_Hand_Enb_state)) - 1 DO
			Response[og_num_counter] := old_Hand_Enb_state[og_i];
			og_num_counter := og_num_counter + 1;
		END_FOR
	END_IF
	
	// Hand enable error state
	IF outrobot_state.Hand_Enb_Err <> old_robot_state.Hand_Enb_Err THEN
		IF outrobot_state.Hand_Enb_Err THEN	// if true
			old_Hand_Enb_Err_state[9] := 49;
		ELSE
			old_Hand_Enb_Err_state[9] := 48;
		END_IF
		
		FOR og_i := 0 TO UDINT_TO_INT(SIZEOF(old_Hand_Enb_Err_state)) - 1 DO
			Response[og_num_counter] := old_Hand_Enb_Err_state[og_i];
			og_num_counter := og_num_counter + 1;
		END_FOR
	END_IF
	
	// hand move error state
	IF outrobot_state.Hand_Mov_Err <> old_robot_state.Hand_Mov_Err THEN
		IF outrobot_state.Hand_Mov_Err THEN	// if true
			old_Hand_Mov_Err_state[9] := 49;
		ELSE
			old_Hand_Mov_Err_state[9] := 48;
		END_IF
		
		FOR og_i := 0 TO UDINT_TO_INT(SIZEOF(old_Hand_Mov_Err_state)) - 1 DO
			Response[og_num_counter] := old_Hand_Mov_Err_state[og_i];
			og_num_counter := og_num_counter + 1;
		END_FOR
	END_IF
	
	// robot move error state
	IF outrobot_state.Robot_Mov_Err <> old_robot_state.Robot_Mov_Err THEN
		IF outrobot_state.Robot_Mov_Err THEN	// if true
			old_Robot_Mov_Err_state[9] := 49;
		ELSE
			old_Robot_Mov_Err_state[9] := 48;
		END_IF
		
		FOR og_i := 0 TO UDINT_TO_INT(SIZEOF(old_Robot_Mov_Err_state)) - 1 DO
			Response[og_num_counter] := old_Robot_Mov_Err_state[og_i];
			og_num_counter := og_num_counter + 1;
		END_FOR
	END_IF
	
	// CNC executing or not
	IF outrobot_state.CNC_Executing <> old_robot_state.CNC_Executing THEN
		IF outrobot_state.CNC_Executing THEN	// if true
			old_CNC_Executing_state[8] := 49;
		ELSE
			old_CNC_Executing_state[8] := 48;
		END_IF
		
		FOR og_i := 0 TO UDINT_TO_INT(SIZEOF(old_CNC_Executing_state)) - 1 DO
			Response[og_num_counter] := old_CNC_Executing_state[og_i];
			og_num_counter := og_num_counter + 1;
		END_FOR
	END_IF
	
	// CNC Error
	IF outrobot_state.CNC_Execute_Err <> old_robot_state.CNC_Execute_Err THEN
		IF outrobot_state.CNC_Execute_Err THEN	// if true
			old_CNC_Err_state[8] := 49;
		ELSE
			old_CNC_Err_state[8] := 48;
		END_IF
		
		FOR og_i := 0 TO UDINT_TO_INT(SIZEOF(old_CNC_Err_state)) - 1 DO
			Response[og_num_counter] := old_CNC_Err_state[og_i];
			og_num_counter := og_num_counter + 1;
		END_FOR
	END_IF
	
	// CNC finish or not
	IF outrobot_state.CNC_Execute_Done <> old_robot_state.CNC_Execute_Done THEN
		IF outrobot_state.CNC_Execute_Done THEN	// if true
			old_CNC_Done_state[9] := 49;
		ELSE
			old_CNC_Done_state[9] := 48;
		END_IF
		
		FOR og_i := 0 TO UDINT_TO_INT(SIZEOF(old_CNC_Done_state)) - 1 DO
			Response[og_num_counter] := old_CNC_Done_state[og_i];
			og_num_counter := og_num_counter + 1;
		END_FOR
	END_IF
	
	(*	templet for new laybel
	// CNC executing or not
	IF outrobot_state. <> old_robot_state. THEN
		IF outrobot_state. THEN	// if true
			[6] := 49;
		ELSE
			[6] := 48;
		END_IF
		
		FOR og_i := 0 TO UDINT_TO_INT(SIZEOF()) - 1 DO
			Response[og_num_counter] := [og_i];
			og_num_counter := og_num_counter + 1;
		END_FOR
	END_IF
	*)
	
	// add ending
	FOR og_i := 0 TO 1 DO
		Response[og_num_counter] := 91;	// [
		og_num_counter := og_num_counter + 1;
		Response[og_num_counter] := data_end[og_i];	// CR, LF
		og_num_counter := og_num_counter + 1;
		Response[og_num_counter] := 93;	// ]
		og_num_counter := og_num_counter + 1;
	END_FOR
	
	Response_Data_Size := INT_TO_UDINT(og_num_counter);
	Response_Valid := TRUE;
	old_robot_state := outrobot_state;
END_IF

END_FUNCTION_BLOCK

// Device/Application/Organize_Hand_Command
FUNCTION_BLOCK Organize_Hand_Command
VAR_INPUT
	enable :BOOL;
	New_Cmd_valid : BOOL;
	new_cmd : robot_command_via_tcp;
	Grab : BOOL;
	Gesture_Valid : BOOL;
	Gesture_Type : INT;
	Enable_Hand : BOOL;
	Demo_Hand : BOOL;
END_VAR
VAR_OUTPUT
	Done : BOOL;
	Current_Hand_State : robot_state;
	Err : BOOL;
	Err_Message : error_message;
END_VAR
VAR
	// internal state
	_enable : BOOL;
	_state : INT; // block state machine
	_next_state : INT;
	_newCMD : BOOL;	// if ready to execute new command
	
	// internal command
	_old_ovr : INT := 40;
	_old_gest : gesture_type; 
	_old_enb_state, _old_grab_state, _old_demo_state : BOOL; 
	_empty_hand_state :  robot_state;	// use to reset out put hand state
	
	// blocks
	Hand_power : Auxaxis_PowerOn;
	Hand_Demo : hand_gesture_demo;
	hand_Gesture : Hand_Gesture;
	_errMessage : error_message;
	
	// debug
END_VAR

IF NOT enable AND _enable THEN	// if turn off and block not yet initialize 
	hand_demo(enable := enable);
	hand_gesture(enable := enable);
	Hand_power(enable := enable);
	_newCMD := err := _enable := FALSE;
	_errMessage := Err_Message := error_message.Err_None;
	_State := 0;
	Current_Hand_State := _empty_hand_state;
	RETURN;
ELSIF NOT enable THEN
	RETURN;
ELSIF enable THEN
	_enable := TRUE;
END_IF

// get new command
IF new_cmd_valid THEN
	IF new_cmd.Enabl_Hand_Valid THEN	// if enable or disable hand
		_newCMD := TRUE;	// new command is come
		_old_enb_state := new_cmd.Enabl_Hand_state;
		_next_state := 10;
	END_IF
	
	IF new_cmd.Gesture_Demo_Valid THEN	// if play demo
		_newCMD := TRUE;
		_old_demo_state := new_cmd.Gesture_Demo_state;
		_next_state := 20;
	END_IF
	
	IF new_cmd.Grab_Valid THEN	// if open or close grab
		_newCMD := TRUE;
		IF new_cmd.Grab_state THEN
			_old_gest := 10;
		ELSE
			_old_gest := 11;
		END_IF
		_next_state := 40;
	END_IF
	
	IF new_cmd.Gesture_Valid THEN	// if ask hand to show one gesture
		_newCMD := TRUE;
		_old_gest := new_cmd.Gesture_Num;
		_next_state := 40;
	END_IF
END_IF

// if try to send movement command but hand is not enabled
IF _state > 10 AND NOT Current_Hand_State.Hand_Enabled THEN
	//_state := -10;
END_IF

CASE (_state) OF 
	-20:
		Current_Hand_State.Hand_Mov_Err := TRUE;
		Err_Message := _errMessage;
		_state := -1;
		
	-10:
		Current_Hand_State.Hand_Enb_Err := TRUE;
		Err_Message := _errMessage;
		_state := -1;
		
	-5:
		IF _errMessage >= 50 AND _errMessage < 80  THEN	// enable err
			_state := -10;
		ELSIF _errMessage >=10 AND _errMessage < 50 THEN // movement err
			_state := -20;
		END_IF
		
	-1:
		IF _newCMD THEN
			Current_Hand_State.Hand_Mov_Err := FALSE;
			Current_Hand_State.Hand_Enb_Err := FALSE;
			_state := 0;
		END_IF
		
	0:
		_newCMD := FALSE;
		_state := _next_state;
		
	10: // enable or disable the hand
		Hand_power(enable := _old_enb_state);
		Current_Hand_State.Hand_Enabled := Hand_power.Done;
		IF hand_power.Error THEN
			_errMessage := hand_power.Err_Message;
			Hand_power(enable := FALSE);	// turn off block after assigned err massage and ready for next enable command
			_state := -5; // enable error
		END_IF
		
		IF _newCMD THEN
			_state := 0;
		END_IF
		
	20:	// start demo gesture
		Hand_Demo(enable:= _old_demo_state, startMov := TRUE, ovr := _old_ovr);
		
		IF Hand_Demo.IsMoving THEN
			Current_Hand_State.Gesture_State := Hand_Demo.Current_Gesture;
		END_IF
		
		IF hand_demo.err THEN
			_errMessage := hand_demo.err_message;
			_state := -5;
		END_IF
		
		IF _newCMD THEN
			Hand_Demo(enable:= FALSE);
			_state := 0;
		END_IF
	
	40:	// show one gesture
		hand_Gesture(enable:= TRUE, overFeed := _old_ovr, gesture := _old_gest);
		IF hand_Gesture.Done AND NOT _newCMD THEN
			Current_Hand_State.Gesture_State := _old_gest;
		END_IF
		IF hand_gesture.Error THEN
			_errmessage := hand_Gesture.Err_Message;
			_state := -5;
		END_IF
		IF _newCMD THEN
			hand_Gesture(enable := FALSE);
			_state := 0;
		END_IF
END_CASE


IF _state < 0 THEN
	err := TRUE;
END_IF

END_FUNCTION_BLOCK

// Device/Application/hand blocks/Hand_Gesture
FUNCTION_BLOCK Hand_Gesture
VAR_INPUT
	Enable : BOOL;
	OverFeed : INT;
	Gesture : Gesture_Type;
END_VAR
VAR_OUTPUT
	Done : BOOL;
	isMoving : BOOL;
	Error : BOOL;
	Err_Message : Error_Message;
END_VAR
VAR
	state : INT := 0;
	i : INT;
	//movment settings
	Finger_Movement: ArcaLibrary.MCAT_MoveDirectAbsolute;
	
	ReadCurrentPos : ArcaLibrary.MC_GroupReadActualPosition;
	CurrPos : ARRAY [1..6] OF REAL;
	CoordSys1: ArcaLibrary.MC_COORD_SYSTEM := mcMCS;
	
	Set1: ArcaLibrary.MCAT_Settings;
	ToolMoveVel:REAL:=100;
	ToolMoveAcc:REAL:=500;
	ToolMoveJrk:REAL:=2500;
	bufmode: ArcaLibrary.MC_BUFFER_MODE:=mcBuffered;
	transition: ArcaLibrary.MC_TRANSITION_MODE:=tmRelativeCornerDistance;
	tmPar: ARRAY [1..12] OF REAL :=[1.0, 1.0, 1.0, 1.0, 1.0, 1.0, 1.0, 1.0, 1.0, 1.0, 1.0, 1.0];

	Pos_For_Hand_Block : ArcaLibrary.MCAT_Position;
	Position_0: ARRAY [1..6] OF REAL :=[0.300, -0.100, 0.200, 160.0, 180.0, 0.0];
	Position_1: ARRAY [1..6] OF REAL :=[0.500, -0.100, 0.200, 160.0, 180.0, 0.0];
	RobotMovPos: ARRAY [1..6] OF REAL :=[0.50, -0.100, 0.200, 160.0, 180.0, 0.0];
	FingerMovPos: ARRAY [1..32] OF REAL;
	SecFingerMovPos: ARRAY [1..32] OF REAL;
	ThdFingerMovPos: ARRAY [1..32] OF REAL;
	CycleMovTimes : INT := 1;
	CycleMovDone : BOOL;
	AxesPosForExternal: ARRAY [1..32] OF REAL;

	Cycle_Movement: ARRAY [1..20] OF ArcaLibrary.MCAT_MoveDirectAbsolute;
	CycleFingerMovPos: ARRAY [1..20] OF ARRAY[1..32] OF REAL;	
	DelayTimer : ton;
	DelayTime : ARRAY [1..20] OF TIME;
	readyToMov : BOOL;
	MaxDifference : REAL := 0.005;
	G_MovObj_Muilt : INT;
	
	// gesture pos
	g_RestPos: ARRAY [1..32] OF REAL;
	g_one: ARRAY [1..32] OF REAL;
	g_two: ARRAY [1..32] OF REAL;
	g_three: ARRAY [1..32] OF REAL;
	g_four: ARRAY [1..32] OF REAL;
	g_five: ARRAY [1..32] OF REAL;
	g_six: ARRAY [1..32] OF REAL;
	g_plam: ARRAY [1..32] OF REAL;
	g_fist: ARRAY [1..32] OF REAL;
	g_thumbUp: ARRAY [1..32] OF REAL;
	g_thumbDown: ARRAY [1..32] OF REAL;
	
	// max degree for every motor
	wrist_0_min : REAL := 0;
	wrist_0_max : REAL := 75;
	wrist_1_min : REAL := 0;
	wrist_1_max : REAL := 75;
	
	thumb_0_min : REAL := 0;
	thumb_0_max : REAL := 70;
	thumb_1_min : REAL := 0;
	thumb_1_max : REAL := 125;
	thumb_2_min : REAL := 0;
	thumb_2_max : REAL := 127;
	thumb_3_min : REAL := 0;
	thumb_3_max : REAL := 127;
	
	index_0_min : REAL := 0;
	index_0_max : REAL := 90;
	index_1_min : REAL := 0;
	index_1_max : REAL := 66;
	index_2_min : REAL := 0;
	index_2_max : REAL := 66;
		
	mid_0_min : REAL := 0;
	mid_0_max : REAL := 60;
	mid_1_min : REAL := 0;
	mid_1_max : REAL := 59;
	mid_2_min : REAL := 0;
	mid_2_max : REAL := 59;
			
	ring_0_min : REAL := 0;
	ring_0_max : REAL := 62;
	ring_1_min : REAL := 0;
	ring_1_max : REAL := 59;
	ring_2_min : REAL := 0;
	ring_2_max : REAL := 59;
		
	little_0_min : REAL := 0;
	little_0_max : REAL := 69;
	little_1_min : REAL := 0;
	little_1_max : REAL := 77;
	little_2_min : REAL := 0;
	little_2_max : REAL := 77;
	
	// debug
END_VAR

IF NOT Enable THEN
	state := 0;
END_IF

IF overfeed > 90 THEN
	overfeed := 90;
ELSIF overfeed < 0 THEN
	overfeed := 0;
END_IF

// read current virtual robot postion
ReadCurrentPos(axesGroup := 0, execute := state > 0, CoordSystem:=mcMcs, Position=>CurrPos);
IF ReadCurrentPos.Error THEN
	state := -10;
END_IF

CASE state OF
	-40:
		error := TRUE;
		Err_Message := error_message.Err_Gesture_Type_Cycle_mov_block_err;
	-30:
		error := TRUE;
		Err_Message := error_message.Err_AuxAxis_Movement_Block_err;
	-20:
		error := TRUE;
		Err_Message := error_message.Err_Gesture_Type_Hand_Pos_Not_Given;
	-10:
	(*
		IF ReadCurrentPos.ErrorID THEN
			
		END_IF
	*)
		error := TRUE;
		Err_Message := error_message.Err_AuxAxis_Movement_Cannot_read_virture_robot_position;
		
	0:
		done := error := FALSE;
		Err_Message := error_message.Err_None;
		
		IF Enable THEN
			IF Gesture <> Gesture_Type.Gesture_Type_none THEN
				state := 10;
			ELSE 
				state := -20;
			END_IF
		END_IF

	10:	//initialize
	
		// set hand pos to relax position
		g_RestPos[1] := (index_0_max - index_0_min)/2 + index_0_min;
		g_RestPos[2] := (index_1_max - index_1_min)/2 + index_1_min;
		g_RestPos[3] := (mid_0_max - mid_0_min)/2 + mid_0_min;
		g_RestPos[4] := (mid_1_max - mid_1_min)/2 + mid_1_min;
		g_RestPos[5] := (ring_0_max - ring_0_min)/2 + ring_0_min;
		g_RestPos[6] := (ring_1_max - ring_1_min)/2 + ring_1_min;
		g_RestPos[7] := (little_0_max - little_0_min)/2 + little_0_min;
		g_RestPos[8] := (little_1_max - little_1_min)/2 + little_1_min;
		g_RestPos[9] := thumb_0_min;
		g_RestPos[10] := thumb_1_min;
		g_RestPos[11] := thumb_2_min;
		g_RestPos[12] := wrist_0_min;
		g_RestPos[13] := wrist_1_min;
		
		g_RestPos[14] := thumb_3_min;
		g_RestPos[15] := index_2_min;
		g_RestPos[16] := mid_2_min;
		g_RestPos[17] := ring_2_min;
		g_RestPos[18] := little_2_min;
		
		//one
		g_one[1]		:= index_0_min;	//	index 0
		g_one[2]		:= index_1_min;	//	index 1
		g_one[3]		:= mid_0_max;	//	mid 0
		g_one[4]		:= mid_1_max;	//	mid 1
		g_one[5]		:= ring_0_max;;	//	ring 0
		g_one[6]		:= ring_1_max;	//	ring 1
		g_one[7]		:= little_0_max;	//	little 0
		g_one[8]		:= little_1_max;	//	little 1
		g_one[9]		:= thumb_0_max;		//	thumb 0
		g_one[10]		:= thumb_1_max;		//	thumb 1
		g_one[11]		:= thumb_2_max;		//	thumb 2
		g_one[12]		:= g_RestPos[12];	// wrist 0
		g_one[13]		:= g_RestPos[13];	// wrist 1
		
		g_one[14] := thumb_3_max;
		g_one[14] := index_2_min;
		g_one[15] := mid_2_min;
		g_one[16] := ring_2_min;
		g_one[17] := little_2_min;
		
		// two
		g_two[1]		:= index_0_min;	//	index 0
		g_two[2]		:= index_1_min;	//	index 1
		g_two[3]		:= mid_0_min;	//	mid 0
		g_two[4]		:= mid_1_min;	//	mid 1
		g_two[5]		:= ring_0_max;;	//	ring 0
		g_two[6]		:= ring_1_max;	//	ring 1
		g_two[7]		:= little_0_max;	//	little 0
		g_two[8]		:= little_1_max;	//	little 1
		g_two[9]		:= thumb_0_max;	//	thumb 0
		g_two[10]		:= thumb_1_max;	//	thumb 1
		g_two[11]		:= thumb_2_max;	//	thumb 2
		g_two[12]		:= g_RestPos[12];	// wrist 0
		g_two[13]		:= g_RestPos[13];	// wrist 1
		
		g_two[14] := thumb_3_max;
		g_two[14] := index_2_min;
		g_two[15] := mid_2_min;
		g_two[16] := ring_2_min;
		g_two[17] := little_2_min;
		
		//three
		g_three[1]		:= index_0_min;	//	index 0
		g_three[2]		:= index_1_min;	//	index 1
		g_three[3]		:= mid_0_min;	//	mid 0
		g_three[4]		:= mid_1_min;	//	mid 1
		g_three[5]		:= ring_0_min;	//	ring 0
		g_three[6]		:= ring_1_min;	//	ring 1
		g_three[7]		:= little_0_max;	//	little 0
		g_three[8]		:= little_1_max;	//	little 1
		g_three[9]		:= thumb_0_max;	//	thumb 0
		g_three[10]		:= thumb_1_max;	//	thumb 1
		g_three[11]		:= thumb_2_max;	//	thumb 2
		g_three[12]		:= g_RestPos[12];	// wrist 0
		g_three[13]		:= g_RestPos[13];	// wrist 1
		
		g_three[14] := thumb_3_max;
		g_three[14] := index_2_min;
		g_three[15] := mid_2_min;
		g_three[16] := ring_2_min;
		g_three[17] := little_2_min;
		
		//four
		g_four[1]		:= index_0_min;	//	index 0
		g_four[2]		:= index_1_min;	//	index 1
		g_four[3]		:= mid_0_min;	//	mid 0
		g_four[4]		:= mid_1_min;	//	mid 1
		g_four[5]		:= ring_0_min;	//	ring 0
		g_four[6]		:= ring_1_min;	//	ring 1
		g_four[7]		:= little_0_min;	//	little 0
		g_four[8]		:= little_1_min;	//	little 1
		g_four[9]		:= thumb_0_max;	//	thumb 0
		g_four[10]		:= thumb_1_max;	//	thumb 1
		g_four[11]		:= thumb_2_max;	//	thumb 2
		g_four[12]		:= g_RestPos[12];	// wrist 0
		g_four[13]		:= g_RestPos[13];	// wrist 1
		
		g_four[14] := thumb_3_max;
		g_four[14] := index_2_min;
		g_four[15] := mid_2_min;
		g_four[16] := ring_2_min;
		g_four[17] := little_2_min;
		
		//five
		g_five[1]		:= index_0_min;	//	index 0
		g_five[2]		:= index_1_min;	//	index 1
		g_five[3]		:= mid_0_min;	//	mid 0
		g_five[4]		:= mid_1_min;	//	mid 1
		g_five[5]		:= ring_0_min;	//	ring 0
		g_five[6]		:= ring_1_min;	//	ring 1
		g_five[7]		:= little_0_min;	//	little 0
		g_five[8]		:= little_1_min;	//	little 1
		g_five[9]		:= thumb_0_min;	//	thumb 0
		g_five[10]		:= thumb_1_min;	//	thumb 1
		g_five[11]		:= thumb_2_min;	//	thumb 2
		g_five[12]		:= g_RestPos[12];	// wrist 0
		g_five[13]		:= g_RestPos[13];	// wrist 1
		
		g_five[14] := thumb_3_min;
		g_five[14] := index_2_min;
		g_five[15] := mid_2_min;
		g_five[16] := ring_2_min;
		g_five[17] := little_2_min;
		
		//six
		g_six[1]		:= index_0_max;	//	index 0
		g_six[2]		:= index_1_max;	//	index 1
		g_six[3]		:= mid_0_max;	//	mid 0
		g_six[4]		:= mid_1_max;	//	mid 1
		g_six[5]		:= ring_0_max;	//	ring 0
		g_six[6]		:= ring_1_max;	//	ring 1
		g_six[7]		:= little_0_min;	//	little 0
		g_six[8]		:= little_1_min;	//	little 1
		g_six[9]		:= thumb_0_min;	//	thumb 0
		g_six[10]		:= thumb_1_min;	//	thumb 1
		g_six[11]		:= thumb_2_min;	//	thumb 2
		g_six[12]		:= g_RestPos[12];	// wrist 0
		g_six[13]		:= g_RestPos[13];	// wrist 1
		
		g_six[14] := thumb_3_min;
		g_six[14] := index_2_min;
		g_six[15] := mid_2_min;
		g_six[16] := ring_2_min;
		g_six[17] := little_2_min;
		
		//plam
		g_plam[1]		:= index_0_min;	//	index 0
		g_plam[2]		:= index_1_min;	//	index 1
		g_plam[3]		:= mid_0_min;	//	mid 0
		g_plam[4]		:= mid_1_min;	//	mid 1
		g_plam[5]		:= ring_0_min;	//	ring 0
		g_plam[6]		:= ring_1_min;	//	ring 1
		g_plam[7]		:= little_0_min;	//	little 0
		g_plam[8]		:= little_1_min;	//	little 1
		g_plam[9]		:= thumb_0_min;	//	thumb 0
		g_plam[10]		:= thumb_1_min;	//	thumb 1
		g_plam[11]		:= thumb_2_min;	//	thumb 2
		g_plam[12]		:= g_RestPos[12];	// wrist 0
		g_plam[13]		:= g_RestPos[13];	// wrist 1
		
		g_plam[14] := thumb_3_min;
		g_plam[14] := index_2_min;
		g_plam[15] := mid_2_min;
		g_plam[16] := ring_2_min;
		g_plam[17] := little_2_min;
		
		//fist
		g_fist[1]		:= index_0_max;	//	index 0
		g_fist[2]		:= index_1_max;	//	index 1
		g_fist[3]		:= mid_0_max;	//	mid 0
		g_fist[4]		:= mid_1_max;	//	mid 1
		g_fist[5]		:= ring_0_max;	//	ring 0
		g_fist[6]		:= ring_1_max;	//	ring 1
		g_fist[7]		:= little_0_max;	//	little 0
		g_fist[8]		:= little_1_max;	//	little 1
		g_fist[9]		:= thumb_0_max;	//	thumb 0
		g_fist[10]		:= thumb_1_max;	//	thumb 1
		g_fist[11]		:= thumb_2_max;	//	thumb 2
		g_fist[12]		:= g_RestPos[12];	// wrist 0
		g_fist[13]		:= g_RestPos[13];	// wrist 1
		
		g_fist[14] := thumb_3_max;
		g_fist[14] := index_2_min;
		g_fist[15] := mid_2_min;
		g_fist[16] := ring_2_min;
		g_fist[17] := little_2_min;
		
		//thumb up
		g_thumbUp[1]		:= index_0_max;	//	index 0
		g_thumbUp[2]		:= index_1_max;	//	index 1
		g_thumbUp[3]		:= mid_0_max;	//	mid 0
		g_thumbUp[4]		:= mid_1_max;	//	mid 1
		g_thumbUp[5]		:= ring_0_max;	//	ring 0
		g_thumbUp[6]		:= ring_1_max;	//	ring 1
		g_thumbUp[7]		:= little_0_max;	//	little 0
		g_thumbUp[8]		:= little_1_max;	//	little 1
		g_thumbUp[9]		:= thumb_0_min;	//	thumb 0
		g_thumbUp[10]		:= thumb_1_min;	//	thumb 1
		g_thumbUp[11]		:= thumb_2_min;	//	thumb 2
		g_thumbUp[12]		:= g_RestPos[12];	// wrist 0
		g_thumbUp[13]		:= g_RestPos[13];	// wrist 1
	
		g_thumbUp[14] := thumb_3_min;
		g_thumbUp[14] := index_2_min;
		g_thumbUp[15] := mid_2_min;
		g_thumbUp[16] := ring_2_min;
		g_thumbUp[17] := little_2_min;
		
		(*	--useless
		//thumb down
		g_thumbDown[1]		:= index_0_max;	//	index 0
		g_thumbDown[2]		:= index_1_max;	//	index 1
		g_thumbDown[3]		:= mid_0_max;	//	mid 0
		g_thumbDown[4]		:= mid_1_max;	//	mid 1
		g_thumbDown[5]		:= ring_0_max;	//	ring 0
		g_thumbDown[6]		:= ring_1_max;	//	ring 1
		g_thumbDown[7]		:= little_0_max;	//	little 0
		g_thumbDown[8]		:= little_1_max;	//	little 1
		g_thumbDown[9]		:= thumb_0_min;	//	thumb 0
		g_thumbDown[10]		:= (thumb_1_max - thumb_1_min)/2 + thumb_1_min;	//	thumb 1
		g_thumbDown[11]		:= thumb_2_min;	//	thumb 2
		g_thumbDown[12]		:= g_RestPos[12];	// wrist 0
		g_thumbDown[13]		:= g_RestPos[13];	// wrist 1
		
		g_thumbDown[14] := index_2_min;
		g_thumbDown[15] := mid_2_min;
		g_thumbDown[16] := ring_2_min;
		g_thumbDown[17] := little_2_min;
		*)
		
		// take a judge to find where is the robot and give a different destination
		IF ABS(CurrPos[1] - Position_0[1]) > MaxDifference THEN
			RobotMovPos := Position_0;
		ELSE 
			RobotMovPos := Position_1;
		END_IF
		
		// asign value for hand movment block
		Pos_For_Hand_Block.Position := RobotMovPos;
		Pos_For_Hand_Block.AxesPosition:=AxesPosForExternal;
		Pos_For_Hand_Block.AuxAxes:=g_RestPos;
		Pos_For_Hand_Block.CoordSystem:=CoordSys1;
		
		Set1.Velocity:=ToolMoveVel;
		Set1.Acceleration:=ToolMoveAcc;
		Set1.Deceleration:=ToolMoveAcc;
		Set1.Jerk:=ToolMoveJrk;
		Set1.OverfeedPerc:=Overfeed;
		Set1.BufferMode:=bufmode;
		Set1.TransitionMode:=transition;
		Set1.TransitionParameter:=tmPar;
		
		Finger_Movement(AxesGroup:=0, Execute:=FALSE);
		State := 20;
	20:
		IF (NOT enable) THEN
			State := 0;
		END_IF
		
		Finger_Movement(AxesGroup:=0, Execute:=TRUE, Position:=Pos_For_Hand_Block, Settings:=Set1, active => isMoving);
		
		IF Finger_Movement.Done THEN
			Finger_Movement(AxesGroup:=0, Execute:=FALSE);
			state := 30;
		ELSIF Finger_Movement.Error OR Finger_Movement.CommandAborted THEN
			state := -30;
		END_IF
	30:
		CycleMovTimes := 1;	// indecate the hand will move how many cycle.
		FOR i := 1 TO 10 DO
			DelayTime[i] := T#0S;
		END_FOR
		
		CASE Gesture OF
			Gesture_Type.Gesture_Type_none:
				state := -20;
				
			Gesture_Type.Gesture_Type_Num_1:
				SecFingerMovPos := FingerMovPos := g_one;
				
				FingerMovPos[9]		:= g_RestPos[9];
				FingerMovPos[10]	:= g_RestPos[10];
				FingerMovPos[11]	:= g_RestPos[11];
				
				CycleMovTimes := 2;
				CycleFingerMovPos[1] := FingerMovPos;
				CycleFingerMovPos[2] := SecFingerMovPos;

			Gesture_Type.Gesture_Type_Num_2:
				SecFingerMovPos := FingerMovPos := g_two;
				
				FingerMovPos[9]		:= g_RestPos[9];
				FingerMovPos[10]	:= g_RestPos[10];
				FingerMovPos[11]	:= g_RestPos[11];
				
				CycleMovTimes := 2;
				CycleFingerMovPos[1] := FingerMovPos;
				CycleFingerMovPos[2] := SecFingerMovPos;

			Gesture_Type.Gesture_Type_Num_3:
				SecFingerMovPos := FingerMovPos := g_three;
				
				FingerMovPos[9]		:= g_RestPos[9];
				FingerMovPos[10]	:= g_RestPos[10];
				FingerMovPos[11]	:= g_RestPos[11];
				
				CycleMovTimes := 2;
				CycleFingerMovPos[1] := FingerMovPos;
				CycleFingerMovPos[2] := SecFingerMovPos;

			Gesture_Type.Gesture_Type_Num_4:
				FingerMovPos := g_four;
				
				CycleFingerMovPos[1] := FingerMovPos;

			Gesture_Type.Gesture_Type_Num_5:
				FingerMovPos := g_five;
				
				CycleFingerMovPos[1] := FingerMovPos;

			Gesture_Type.Gesture_Type_Num_6:
				FingerMovPos := g_six;
				
				CycleFingerMovPos[1] := FingerMovPos;

			Gesture_Type.Gesture_Type_Fist:
				SecFingerMovPos := FingerMovPos := g_fist;
				
				FingerMovPos[9]		:= g_RestPos[9];
				FingerMovPos[10]	:= g_RestPos[10];
				FingerMovPos[11]	:= g_RestPos[11];
				
				//CycleMovTimes := 2;
				//CycleFingerMovPos[1] := FingerMovPos;
				//CycleFingerMovPos[2] := SecFingerMovPos;
				CycleFingerMovPos[1] := SecFingerMovPos;
				
			Gesture_Type.Gesture_Type_Palm:
				FingerMovPos := g_plam;
				
				CycleFingerMovPos[1] := FingerMovPos;
				
			Gesture_Type.Gesture_Type_ThumbDown:
				FingerMovPos := g_thumbdown;
				
				CycleFingerMovPos[1] := FingerMovPos;
				
			Gesture_Type.Gesture_Type_ThumbUp:
				FingerMovPos := g_thumbup;
				
				CycleFingerMovPos[1] := FingerMovPos;
				
			Gesture_Type.Gesture_Type_ComeOnBaby:
			
				ThdFingerMovPos := SecFingerMovPos := FingerMovPos := g_one;
				
				SecFingerMovPos[1] := g_RestPos [1];
				SecFingerMovPos[2] := index_1_max;
				
				FingerMovPos[9]		:= g_RestPos[9];
				FingerMovPos[10]	:= g_RestPos[10];
				FingerMovPos[11]	:= g_RestPos[11];
				
				CycleMovTimes := 9;
				CycleFingerMovPos[1] := FingerMovPos;
				FOR i := 2 TO CycleMovTimes DO
					IF (i MOD 2) = 1 THEN
						CycleFingerMovPos[i] := SecFingerMovPos;
					ELSE
						CycleFingerMovPos[i] := ThdFingerMovPos;
					END_IF
				END_FOR
				
			Gesture_Type.Gesture_Type_PointTo:
				SecFingerMovPos := FingerMovPos := g_one;
				
				FingerMovPos[9]		:= g_RestPos[9];
				FingerMovPos[10]	:= g_RestPos[10];
				FingerMovPos[11]	:= g_RestPos[11];
				
				//SecFingerMovPos[12] := wrist_0_max;
				//SecFingerMovPos[13] := wrist_1_max;
				
				CycleMovTimes := 2;
				CycleFingerMovPos[1] := FingerMovPos;
				CycleFingerMovPos[2] := SecFingerMovPos;
				
			Gesture_Type.Gesture_Type_Wave:
			
				SecFingerMovPos := FingerMovPos	:= g_two;
				
				FingerMovPos[12] := wrist_0_min;
				FingerMovPos[13] := wrist_1_max;
				
				SecFingerMovPos[13] := - wrist_1_max;
				
				CycleMovTimes := 8;
				FOR i := 1 TO CycleMovTimes DO
					IF (i MOD 2) = 1 THEN
						CycleFingerMovPos[i] := FingerMovPos;
					ELSE
						CycleFingerMovPos[i] := SecFingerMovPos;
					END_IF
				END_FOR
					
			Gesture_Type.Gesture_Type_Nya:
			
				SecFingerMovPos := FingerMovPos	:= g_fist;
				
				FingerMovPos[12] := wrist_0_max;
				FingerMovPos[13] := wrist_1_min;
				
				SecFingerMovPos[12] := - wrist_0_max;
				
				CycleMovTimes := 8;
				FOR i := 1 TO CycleMovTimes DO
					IF (i MOD 2) = 1 THEN
						CycleFingerMovPos[i] := FingerMovPos;
					ELSE
						CycleFingerMovPos[i] := SecFingerMovPos;
					END_IF
				END_FOR
				
			Gesture_Type.Gesture_Type_MovObj:
			
				G_MovObj_Muilt := 2;
				FingerMovPos	:= g_plam;
				SecFingerMovPos	:= g_fist;
				CycleMovTimes := 0;	// initialize
				
				CycleMovTimes := CycleMovTimes + 1;
				FingerMovPos[12] := -wrist_0_max;
				FingerMovPos[13] := wrist_1_max;
				// first mov, hand release go up left
				CycleFingerMovPos[CycleMovTimes] := FingerMovPos;
				//---
				
				CycleMovTimes := CycleMovTimes + 1;
				FingerMovPos[12] := wrist_0_max / G_MovObj_Muilt;
				FingerMovPos[13] := wrist_1_max;
				// sec mov, hand release go down left
				CycleFingerMovPos[CycleMovTimes] := FingerMovPos;
				//---
				
				CycleMovTimes := CycleMovTimes + 1;
				SecFingerMovPos[12] := wrist_0_max  / G_MovObj_Muilt;;
				SecFingerMovPos[13] := wrist_1_max;
				// third mov, hand grab at down left
				CycleFingerMovPos[CycleMovTimes] := SecFingerMovPos;
				//---
				
				CycleMovTimes := CycleMovTimes + 1;
				SecFingerMovPos[12] := -wrist_0_max;
				SecFingerMovPos[13] := wrist_1_max;
				// 4 mov, hand grab go up left
				CycleFingerMovPos[CycleMovTimes] := SecFingerMovPos;
				//---
				
				CycleMovTimes := CycleMovTimes + 1;
				SecFingerMovPos[12] := -wrist_0_max;
				SecFingerMovPos[13] := -wrist_1_max;
				// 5 mov, hand grab go up right
				CycleFingerMovPos[CycleMovTimes] := SecFingerMovPos;
				//---
				
				CycleMovTimes := CycleMovTimes + 1;
				SecFingerMovPos[12] := wrist_0_max / G_MovObj_Muilt;;
				SecFingerMovPos[13] := -wrist_1_max;
				// 6 mov, hand grab go down right
				CycleFingerMovPos[CycleMovTimes] := SecFingerMovPos;
				//---
				
				CycleMovTimes := CycleMovTimes + 1;
				FingerMovPos[12] := wrist_0_max / G_MovObj_Muilt;;
				FingerMovPos[13] := -wrist_1_max;
				// 7 mov, hand release at down right
				CycleFingerMovPos[CycleMovTimes] := FingerMovPos;
				//---
				
				CycleMovTimes := CycleMovTimes + 1;
				FingerMovPos[12] := -wrist_0_max;
				FingerMovPos[13] := -wrist_1_max;
				// 8 mov, hand release go up right
				DelayTime[CycleMovTimes] := T#3S;
				CycleFingerMovPos[CycleMovTimes] := FingerMovPos;
				//---
				
				CycleMovTimes := CycleMovTimes + 1;
				FingerMovPos[12] := wrist_0_max / G_MovObj_Muilt;;
				FingerMovPos[13] := -wrist_1_max;
				// 9 mov, hand release go down right
				CycleFingerMovPos[CycleMovTimes] := FingerMovPos;
				//---
				
				CycleMovTimes := CycleMovTimes + 1;
				SecFingerMovPos[12] := wrist_0_max / G_MovObj_Muilt;;
				SecFingerMovPos[13] := -wrist_1_max;
				// 10 mov, hand grab at down right
				CycleFingerMovPos[CycleMovTimes] := SecFingerMovPos;
				//---
				
				CycleMovTimes := CycleMovTimes + 1;
				SecFingerMovPos[12] := -wrist_0_max;
				SecFingerMovPos[13] := -wrist_1_max;
				// 11 mov, hand grab go up right
				CycleFingerMovPos[CycleMovTimes] := SecFingerMovPos;
				//---
				
				CycleMovTimes := CycleMovTimes + 1;
				SecFingerMovPos[12] := -wrist_0_max;
				SecFingerMovPos[13] := wrist_1_max;
				// 12 mov, hand grab go up left
				CycleFingerMovPos[CycleMovTimes] := SecFingerMovPos;
				//---
				
				CycleMovTimes := CycleMovTimes + 1;
				SecFingerMovPos[12] := wrist_0_max / G_MovObj_Muilt;;
				SecFingerMovPos[13] := wrist_1_max;
				// 13 mov, hand grab at down left
				CycleFingerMovPos[CycleMovTimes] := SecFingerMovPos;
				//---
				
				CycleMovTimes := CycleMovTimes + 1;
				FingerMovPos[12] := wrist_0_max / G_MovObj_Muilt;;
				FingerMovPos[13] := wrist_1_max;
				// 14 mov, hand release at down left
				CycleFingerMovPos[CycleMovTimes] := FingerMovPos;
				//---
		END_CASE
		
		// take a judge to find where is the robot and give a different destination
		IF ABS(CurrPos[1] - Position_0[1]) > MaxDifference THEN
			Pos_For_Hand_Block.Position := Position_0;
		ELSE 
			Pos_For_Hand_Block.Position := Position_1;
		END_IF
		
		// prepare movement block
		FOR i:=1 TO 10 DO
			Cycle_Movement[i](Axesgroup := 0, Execute:=FALSE);
		END_FOR
		
		i := 1;
		Pos_For_Hand_Block.AuxAxes := CycleFingerMovPos [i];
		Set1.OverfeedPerc := Overfeed;
		
		state := 40;
		
	40:
		IF (NOT enable) THEN
			State := 0;
		END_IF
		
		Set1.OverfeedPerc := Overfeed;
		Cycle_Movement[i](AxesGroup:=0, Execute:=TRUE, Position:=Pos_For_Hand_Block, Settings:=Set1, active => isMoving);
		
		IF Cycle_Movement[i].Done THEN
			IF DelayTime[i] > T#0S AND NOT DelayTimer.Q THEN
				DelayTimer(in := TRUE, pt := DelayTime[i]);
			ELSE
				DelayTimer(in := FALSE);
				i := i + 1;
				Pos_For_Hand_Block.AuxAxes := CycleFingerMovPos [i];
				// take a judge to find where is the robot and give a different destination
				IF ABS(CurrPos[1] - Position_0[1]) > MaxDifference THEN
					Pos_For_Hand_Block.Position := Position_0;
				ELSE 
					Pos_For_Hand_Block.Position := Position_1;
				END_IF
			END_IF
		ELSIF Finger_Movement.Error OR Finger_Movement.CommandAborted THEN
			state := -40;
		END_IF
		
		IF i > CycleMovTimes THEN
			state := 50;
		END_IF
	50:
		done := TRUE;
END_CASE
// end of the program

END_FUNCTION_BLOCK

// Device/Application/hand blocks/AuxAxis_PowerOn
FUNCTION_BLOCK AuxAxis_PowerOn
VAR_INPUT
	Enable : BOOL;
END_VAR
VAR_OUTPUT
	Done : BOOL;
	Error : BOOL;
	Err_Message : Error_Message;
END_VAR
VAR
	_state : INT := 0;
	_end : BOOL := TRUE;
	_Timer: ton;
	_err_time : TIME := T#5S;
	
	// read cfg message
	ReadCfg : ArcaLibrary.SYS_GetConfigInfo;
	Num_of_Axis:WORD;
	Num_of_Groups:WORD;
	Num_of_Cams:WORD;
	MotionCfgOK: BOOL;
	ECatCfgOk: BOOL;
	VisionCfgOk: BOOL;
	
	// power settings
	PowBlk:ARRAY[1..48] OF ArcaLibrary.MC_Power;
	PowDone, PowErr: ARRAY [1..48] OF BOOL;
	power_On_States : INT := 0;
	All_Power_On_Check_Counter : INT;
	Power_Err_Check_Counter : INT;
	Power_Counter : INT;
	
	//reset blocks
	AxRes:ARRAY[1..48] OF ArcaLibrary.MC_Reset;
	AxResDone, AxResErr: ARRAY [1..48] OF BOOL;
	rest_counter : INT := 0;
	All_reset_On : BOOL;
	All_reset_On_Check_Counter : INT;
	reset_Err_Check_Counter : INT;
	reset_State : INT := 0;
	
	//group management
	GrpEn: ARRAY[1..5] OF ArcaLibrary.MC_GroupEnable;
	GrpDis: ARRAY[1..5] OF ArcaLibrary.MC_GroupDisable;
	GrpErr : ARRAY [1..5] OF BOOL;
	Grp_En_State : INT;
	Grp_counter : INT;
	Grp_En_Check_Counter : INT;
	Grp_Dis_Counter : INT;
	
	//debug
END_VAR

IF enable  THEN
	_end := FALSE;
ELSE
	_state := -10;
END_IF

IF _end = TRUE THEN
	RETURN;
END_IF

_Timer(in:= (power_On_States = 10) OR (reset_State = 10) OR (Grp_En_State = 10), pt:= _err_time);

// read how many axis has been config
ReadCfg(axisnumber => Num_of_axis, groupnumber => Num_of_Groups, cameranumber => Num_of_Cams
	, MotionCfgOk => MotionCfgOK, ecatcfgok => ECatCfgOk, visioncfgok => VisionCfgOk);

// power blocks
CASE (power_On_States) OF
	0:	
		IF (_state>0 AND _state<100) AND ECatCfgOk AND MotionCfgOK THEN
			power_On_States := 10;
		END_IF
	10:
		All_Power_On_Check_Counter := 1;
		FOR Power_Counter:=1 TO WORD_TO_INT(Num_of_axis) DO
			PowBlk[Power_Counter](Axis:=Power_Counter -1, Enable:=TRUE, EnablePositive:=TRUE, EnableNegative:=TRUE, Status=>PowDone[Power_Counter], Error=>PowErr[Power_Counter]);
			IF PowDone[Power_Counter] = TRUE THEN
				All_Power_On_Check_Counter := All_Power_On_Check_Counter + 1;
			END_IF
		END_FOR
		
		IF All_Power_On_Check_Counter >= WORD_TO_INT(Num_of_axis) THEN
			power_On_States := 20;
		ELSIF _Timer.Q THEN
			_state := -21;
		END_IF
		IF (_state<=0 OR _state>=100) THEN
			power_On_States := 30;
		END_IF
	20:
		IF (_state<=0 OR _state>=100) THEN
			power_On_States := 30;
		END_IF
	30:
		FOR Power_Counter:=1 TO WORD_TO_INT(Num_of_axis) DO
			PowBlk[Power_Counter](Axis:=Power_Counter -1, Enable:=FALSE);
		END_FOR
		power_On_States := 0;
END_CASE
// check if power block is err
IF power_On_States > 0 AND power_On_States < 30 THEN
	FOR Power_Err_Check_Counter:=1 TO WORD_TO_INT(Num_of_axis) DO
			IF PowBlk[Power_Err_Check_Counter - 1].Error = TRUE THEN
				//_state := -20;
			END_IF
	END_FOR
END_IF

// reset blocks
CASE (reset_State) OF
	0:
		All_reset_On := FALSE;
		IF _state=2 THEN
			reset_state := 10;
		END_IF
	10:
		All_reset_On_Check_Counter := 0;
		FOR rest_counter:=1 TO WORD_TO_INT(Num_of_axis) DO
			AxRes[rest_counter](Axis:=rest_counter - 1, Execute:=TRUE, Done=>AxResDone[rest_counter], Error=>AxResErr[rest_counter]);
			IF AxRes[rest_counter].Done = TRUE THEN
				All_reset_On_Check_Counter := All_reset_On_Check_Counter +1;
			END_IF
		END_FOR
		IF All_reset_On_Check_Counter = WORD_TO_INT(Num_of_axis) THEN
			All_reset_On := TRUE;
		ELSIF _Timer.Q THEN
			_state := -31;
		END_IF
		IF (_state <> 2) THEN
			reset_State := 0;
		END_IF
END_CASE
// check if reset block is err
IF reset_State <> 0 THEN
	FOR reset_Err_Check_Counter:=1 TO WORD_TO_INT(Num_of_axis) DO
			IF AxRes[reset_Err_Check_Counter - 1].Error = TRUE THEN
				_state := -30;
			END_IF
	END_FOR
END_IF

// group enable/disable
CASE Grp_En_State OF
	0:
		IF _state >= 30 AND _state <=100 THEN
			grp_counter := 1;
			Grp_En_State := 10;
		END_IF
	10:	
		GrpEn[grp_counter](AxesGroup := grp_counter - 1, Execute := TRUE);
		IF GrpEn[grp_counter].Done THEN
			IF grp_counter <= WORD_TO_INT(Num_of_Groups) THEN
				grp_counter := grp_counter +1;
			END_IF
			IF grp_counter > WORD_TO_INT(Num_of_Groups) THEN
				Grp_En_State := 20;
			END_IF
		ELSIF _Timer.Q THEN
			_state := -41;
		END_IF
		
		IF (_state < 30 OR _state > 100) THEN
			Grp_En_State := 30;
		END_IF
	20:
		IF (_state < 30 OR _state > 100) THEN
			Grp_En_State := 30;
		END_IF
	30:
		FOR grp_counter := 1 TO WORD_TO_INT(Num_of_Groups) DO
			GrpEn[grp_counter](AxesGroup := grp_counter - 1, Execute := FALSE);
		END_FOR
		Grp_En_State := 0;
	
END_CASE
// check if enable block is err
IF Grp_En_State = 9990 THEN
	FOR Grp_En_Check_Counter:=1 TO WORD_TO_INT(Num_of_Groups) DO
			IF GrpEn[Grp_En_Check_Counter - 1].Error = TRUE THEN
				_state := -40;
			END_IF
	END_FOR
END_IF

// disable group when all group enable block are off
FOR Grp_Dis_Counter := 1 TO WORD_TO_INT(Num_of_Groups) DO
	GrpDis[Grp_Dis_Counter](AxesGroup:= Grp_Dis_Counter - 1, Execute:= Grp_En_State = 0);
END_FOR

//	manager
CASE _state OF
	-41:
		error := TRUE;
		err_message := Error_Message.Err_Group_Enable_TimeOut;
	-40:
		error := TRUE;
		err_message := Error_Message.Err_Group_Enable_Block_Err;
		
	-31:
		error := TRUE;
		err_message := Error_Message.Err_Power_Reset_TimeOut;
	-30:
		error := TRUE;
		err_message := Error_Message.Err_Power_Reset_Block_Err;
		
	-21:
		error := TRUE;
		err_message := Error_Message.Err_PowerOn_TimeOut;
	-20:
		error := TRUE;
		err_message := Error_Message.Err_PowerOn_Block_Err;
	-10:
		IF power_On_States = 0 AND reset_State = 0 AND Grp_En_State = 0 THEN
			AllAxisGroupEnb := done := error := FALSE;
			err_message := error_message.Err_None;
			_end := TRUE;
			_state := 0;
		END_IF
	0:
		IF enable AND power_On_States = 0 AND reset_State = 0 AND Grp_En_State = 0 THEN
			_state := 10;
		END_IF
	10:
		IF power_On_States = 20 THEN
			_state := 30;
		END_IF
	30:
		IF Grp_En_State = 20 THEN
			_state := 40;
		END_IF
	40:
		AllAxisGroupEnb := done := TRUE;
END_CASE

END_FUNCTION_BLOCK

// Device/Application/hand blocks/Hand_Gesture_Demo
FUNCTION_BLOCK Hand_Gesture_Demo
VAR_INPUT
	enable :BOOL;
	internal_hand_enable : BOOL;
	startMov :BOOL;
	ovr : INT;
END_VAR

VAR_OUTPUT
	IsEnabled : BOOL;
	IsMoving : BOOL;
	Current_Gesture : Gesture_type;
	err : BOOL;
	err_message : error_message;
END_VAR

VAR
	// state control
	cycleState : INT;	// state machine
	cycleCounter : INT;	// counte how many time already been done
	start_cycle : INT := 1;	// start cycle from a number
	total_cycle_time : INT := 12; //	max cycle time
	cycleTimer : ton;
	cycleDelayTime : TIME := T#2S;	// delay time between every gesture
	
	// hand powerOn
	powerHand : BOOL;
	powerOnHand : AuxAxis_PowerOn;
	_enabled : BOOL;
	
	// gestrure mov block
	GestureMov : Hand_Gesture;
	GestureType : ARRAY [1..16] OF Gesture_type;
END_VAR

// set gesture type
GestureType[1] := Gesture_type.Gesture_Type_Num_1;
GestureType[2] := Gesture_type.Gesture_Type_Num_2;
GestureType[3] := Gesture_type.Gesture_Type_Num_3;
GestureType[4] := Gesture_type.Gesture_Type_Num_4;
GestureType[5] := Gesture_type.Gesture_Type_Num_5;
GestureType[6] := Gesture_type.Gesture_Type_Num_6;
GestureType[7] := Gesture_type.Gesture_Type_Fist;
GestureType[8] := Gesture_type.Gesture_Type_Palm;
GestureType[9] := Gesture_type.Gesture_Type_ThumbUp;
//GestureType[10] := Gesture_type.Gesture_Type_ThumbDown;
GestureType[10] := Gesture_type.Gesture_Type_ComeOnBaby;
//GestureType[11] := Gesture_type.Gesture_Type_PointTo;
GestureType[11] := Gesture_type.Gesture_Type_wave;
GestureType[12] := Gesture_type.Gesture_Type_nya;
GestureType[13] := Gesture_type.Gesture_Type_MovObj;

//err
IF powerOnHand.Error OR GestureMov.Error THEN
	err := TRUE;
	IF powerOnHand.Error THEN
		err_message := powerOnHand.Err_Message;
	ELSIF GestureMov.Error THEN
		err_message := GestureMov.Err_Message;
	END_IF
ELSE
	err := FALSE;
	err_message := error_message.Err_None;
END_IF

// enable hand
IF internal_hand_enable THEN
	powerOnHand(enable := enable);
	_enabled := IsEnabled := powerOnHand.Done;
END_IF

IF NOT enable THEN
	cycleState := 0;
	isMoving := FALSE;
	cycleTimer(in := FALSE);	// reset timer
	GestureMov(Enable := FALSE);	// reset movement block
END_IF

CASE cycleState OF
	0: 
		// if block is enabled and order to move and (manager by internal power or by external power)
		IF enable AND startMov AND (NOT internal_hand_enable OR _enabled) THEN
			cycleCounter := start_cycle;	// set counter to start_cycle for gesture
			cycleState := 10;
		END_IF
	10:
		GestureMov(Enable := TRUE, overfeed := ovr, Gesture := Current_Gesture := GestureType[cycleCounter], isMoving => isMoving);
		IF GestureMov.Done THEN
			cycleTimer(in := TRUE, pt:= cycleDelayTime);	// start timer for delay
			IF cycleTimer.Q THEN	// time reach
				cycleCounter := cycleCounter + 1;	// done and self add for next gesture
				cycleTimer(in := FALSE);	// reset timer
				GestureMov(Enable := FALSE);	// reset movement block
				IF cycleCounter <= total_cycle_time THEN
					cycleState := 10;	// if not reach total number then go back keep do next gesture
				ELSE
					cycleState := 0;	// if reach maximum then go back beginning
				END_IF
			END_IF
		END_IF
		
END_CASE

END_FUNCTION_BLOCK

// Device/Application/CNC Execute/CNC_Execute_Manager
FUNCTION_BLOCK CNC_Execute_Manager
VAR_INPUT
	Enable : BOOL;
	Mov_Group : INT;
	TCP_CMD_Valid : BOOL;
	TCP_CMD : robot_command_via_tcp;
END_VAR
VAR_OUTPUT
	CNC_state : robot_state;
	Done :BOOL;
	Error : BOOL;
	Err_Msg : cnc_error;
END_VAR
VAR
	_enb : BOOL;
	_newCMD : BOOL;
	_oldNum : INT;
	state : INT;
	program_head : STRING := 'PLC_Execute_Hand_Movement.tt/Pos_';
	program_end : STRING := 'sss';
	program_name : STRING;
	
	CNC_Execute : Cnc_KemroExecute;
	timer : ton;
	delay_check : TIME := T#1S;
	debug: INT := 1;
END_VAR

IF Enable THEN
	_enb := TRUE;
ELSIF NOT Enable AND _enb THEN
	_enb := FALSE;
	state := 0;
END_IF

IF TCP_CMD_Valid AND TCP_CMD.CNC_Mov_Valid THEN
	_newCMD := TRUE;
	state := 0;
	_oldNum := TCP_CMD.CNC_Mov_Program_Num;
END_IF

CASE state OF
	-10:
		error := TRUE;
		CASE cnc_execute.ErrorID OF
			0:
				err_msg := 0;
			1:
				err_msg := 1;
			2:
				err_msg := 2;
			3:
				err_msg := 3;
			4:
				err_msg := 4;
			5:
				err_msg := 5;
		END_CASE
	0:
		error := FALSE;
		Err_Msg := 0;
		Done := 0;
		CNC_Execute(axesGroup := mov_group, enable := FALSE, execute := FALSE);
		IF _enb THEN
			state := 10;
		END_IF
	10:
		IF _newCMD THEN
			_newCMD := FALSE;
			// empty the program name first
			program_name := delete(str := program_name, LEN := len(program_name), pos := 1);
			program_name := concat(program_head, INT_TO_STRING(_oldNum));	// give name for plc to execute
			//program_name := concat(program_head, INT_TO_STRING(debug));	// give name for plc to execute
			timer(in:= FALSE);
			state := 20;
		END_IF
	20:
		// check if the program exist
		// if there are no shuch program, plc collapse anyway
		CNC_Execute(axesgroup := Mov_Group, enable := TRUE, programName := program_name);
		timer(in:= TRUE, pt := delay_check);
		IF CNC_Execute.Ready THEN
			state := 30;
		ELSIF cnc_execute.Error THEN
			state := -10;
		ELSIF timer.Q THEN
			state := -10;
		END_IF
	30:
		CNC_Execute(axesgroup := Mov_Group, enable := TRUE, programName := program_name
					, execute := TRUE);
		IF CNC_Execute.Error THEN
			state := -10;
		ELSIF cnc_execute.Done THEN
			state := 40;
		END_IF
	40:
		done := TRUE;
END_CASE

cnc_state.CNC_Executing := CNC_Execute.Busy;
cnc_state.CNC_Execute_Done := cnc_execute.Done;
cnc_state.CNC_Execute_Err := CNC_Execute.Error;

END_FUNCTION_BLOCK

// Device/Application/Vision Control/Vision_Control
FUNCTION_BLOCK Vision_Control
VAR_INPUT
	enable : BOOL;
	cam_id : INT;
	robot_group : INT;
	execute : BOOL;
	delay_pick_obj : TIME;
	wait_signal_before_pick : BOOL;
	isPicked : BOOL;
	delay_release_obj : TIME;
END_VAR
VAR_OUTPUT
	ready : BOOL;
	waitting_for_obj : BOOL;
	ready_to_pick : BOOL;
	ready_to_release : BOOL;
	error : BOOL;
END_VAR
VAR
	State:INT :=0;

	//SERVER
	IPAddr: ArcaLibrary.NBS.IP_ADDR := (sAddr := '192.168.80.100'); //Camera IP address
	Port: UINT :=50010; //camera TCP/IP port

	//TCP-IP camera connection
	TCP_IP_Camera1: ArcaLibrary.PLC_TcpIpCamera;
	ObjDetected: INT:=0;
	ConnectionError, CameraError, WrongWaitCycle: BOOL;
	TimeOut: UDINT:= 10000000;

	//OBJECTS DATA
	ObjList : ARRAY [0..31] OF ArcaLibrary.Vision_ObjectData;
	indexLast : INT; //index for queue scrolling
	i,j,k:INT; //loop counters
	OQueue: ARRAY [0..31] OF ArcaLibrary.PLC_ObjectData;
	OQueue_Prod: INT:=0;
	OQueue_Cons: INT :=0;

	//TIMER
	GetTime:SYS_GetActualTime_U32;
	CurrentTime: UDINT;
	TimeDelay : UDINT := 500000; //delay between two camera iterations [us]
	//Check Objects
	Tolerance:REAL:=18; //given from Reference manual table

	//GetCameraData block
	GetCameraData1: ArcaLibrary.PLC_GetCameraData;
	GetDataDone: BOOL:= FALSE;
	GetDataTrigger: BOOL :=FALSE;
	camerEnb : BOOL;

	// block to switch on axis and group
	PowFb : Auxaxis_Poweron;
	PowEn : BOOL;
	PowError, PowReady:BOOL;

	//BELT
	zeroPCS : ARRAY [0..5] OF REAL;
	BeltPcsFb:ArcaLibrary.MCAT_GroupSetPCS;

	// vacuum valve
	EvFb : BMET_Write_DO;
	Ev: UINT := 0;

	//group move FB
	GrMoveFb1, GrMoveFb2, GrMoveFb3, GrMoveFb4, GrMoveFb5, GrMoveFb6, GrMoveFb7, GrMoveFb8: ArcaLibrary.MC_MoveLinearAbsolute;
	GrMoveFb0 : ArcaLibrary.MCAT_MoveDirect;
	GrMoveFb0_Lin : ArcaLibrary.MC_MoveLinearAbsolute;
	ObjPosUp : ARRAY[1..6] OF REAL := [0.0, 0.0, 0.0, 0.0, 0.0, 0.0];
	ObjPosDown : ARRAY[1..6] OF REAL := [0.0, 0.0, 0.0, 0.0, 0.0, 0.0];
	GrMoveDone, GrMoveDone2, GrMoveDone3, GrMoveDone4: BOOL;
	buff_mod: ArcaLibrary.MC_BUFFER_MODE:= mcBuffered;
	GrRelCorner :REAL := 0.5;
	GrReadPosFb: ArcaLibrary.MC_GroupReadActualPosition;
	GrPosValue: ARRAY [1..6] OF REAL;
	GrStop: ArcaLibrary.MC_GroupHalt;
	OutStop: ArcaLibrary.MC_GroupStop;
	outHalt: ArcaLibrary.MC_GroupHalt;
	outExecute, outHaltDone, outStopDone, outDone2 : BOOL;
	outHaltErr, outStopErr : BOOL;
	safepoint_overfeed : INT := 3;
	RobotSpeed : REAL := 0.05;
	RobotAccel : REAL := 0.15;
	
	//position at begain
	safe_pos : ARRAY [1..6] OF REAL := [0, 0, 0, 0, -90, 0];
	
	// Marker position
	RobotZDelta : REAL := -0.05;
	MarkerUp : ARRAY [1..6] OF REAL := [0.22, -0.3, 0.32, 180.0, 180.0, 0.0];
	MarkerDown : ARRAY [1..6] OF REAL := [0.22, -0.3, 0.31, 180.0, 180.0, 0.0];
	
	// Watting position
	WaittingUp : ARRAY [1..6] OF REAL := [0.345, 0, 0.4, 180.0, 180.0, 0.0];

	//robot position management
	y_entry_bound: REAL:=200;
	y_exit_bound: REAL:=-100;
	Z : REAL := -0.305;
	pos: REAL; //check the X position
	ObjCount: INT;
	AdditionalCompensation: ARRAY [1..3] OF REAL := [0.0, 0.0, 0.0]; //additional tracking error compensation

	// 103 error restart
	err103_counter : INT;
	err103state : INT;
	err103_timer : ton;
	
	//DEBUG
	NextObjPos, NextObjPosX: REAL;
	CameraObjN: INT;
	RobX, RobY: REAL;
	PickTimer : ton;
	
	testReal : ARRAY [1..12] OF REAL;
	debugButton : BOOL := TRUE;
	debugButton_2 : BOOL;
	debugButton_3 : BOOL;
	debugButton_4 : BOOL;
	delayTime : TIME := T#500MS;
	_def_delayTime : TIME := T#500MS;
	debug_Pos:REAL;
	
	debugLook : BOOL;
	
	debugkkk : BOOL;
	debugbbb : BOOL;
END_VAR

(* Debug function

RETURN;
*)
IF delay_pick_obj <> T#0S THEN
	delayTime := delay_pick_obj;
ELSE
	delayTime := _def_delayTime;
END_IF

//Get time and power on FB
GetTime(Enable:=TRUE, ActualTime=>CurrentTime);
PowFb(enable:= State > 0 AND state <= 80, done => PowReady, Error=>PowError);

//handle TCP-IP connection to the camera

TCP_IP_Camera1(Enable:=camerEnb, Start:=execute, IpAddress:=IPAddr, Port:=Port, ConnectionTimeout:=TimeOut, CameraID:=cam_id, 
	TimeDelay:=TimeDelay, CurrentTime:=CurrentTime, GetDataDone:=GetDataDone, 
	BeltActualPos:= 0, ObjList=>ObjList, ObjDetected=>ObjDetected, indexLast=>indexLast, 
	GetDataTrigger=>GetDataTrigger, ConnectionError=>ConnectionError, CameraError=>CameraError, 
	WrongWaitCycle=>WrongWaitCycle);

	
//Data evaluation
GetCameraData1(ObjList:=ADR(ObjList), ObjDetected:=ObjDetected, indexLast:=indexLast, BeltSpeed:=0, BeltActualPos:=0,
	BeltDirection:=2, ToleranceValue:= Tolerance, Enable:=debugLook(*Enable*), GetDataTrigger:=GetDataTrigger, CurrentTime:=CurrentTime, OQueue=>OQueue,
	OQueue_Prod=>OQueue_Prod, GetDataDone=>GetDataDone);
	
// Read measures
GrReadPosFb(AxesGroup:=robot_group, CoordSystem:=mcMcs, Execute:=State>0, Position=>GrPosValue);
RobX:= GrPosValue[1];
RobY:= GrPosValue[2];

// PCS UPDATE
// NOTE: Belt is moving in the X direction in the OPPOSITE WAY to robot
IF (State>2) THEN
	IF OQueue_Prod <> OQueue_Cons THEN
		OQueue[OQueue_Cons].CurrPos[1] := OQueue[OQueue_Cons].DetectPos[1] + AdditionalCompensation[1];
		OQueue[OQueue_Cons].CurrPos[2] := OQueue[OQueue_Cons].DetectPos[2] + AdditionalCompensation[2];
		OQueue[OQueue_Cons].CurrPos[3] := 0.0;
		IF debugButton THEN
			OQueue[OQueue_Cons].CurrPos[4] := 180;
			OQueue[OQueue_Cons].CurrPos[5] := 180;
			OQueue[OQueue_Cons].CurrPos[6] := 0; //OQueue[OQueue_Cons].DetectPos[6];
		ELSE
			OQueue[OQueue_Cons].CurrPos[4] := 180;
			OQueue[OQueue_Cons].CurrPos[5] := 180;
			OQueue[OQueue_Cons].CurrPos[6] := 0;
		END_IF
		BeltPcsFb(AxesGroup:=robot_group, Enable:=TRUE, PcsPos:=OQueue[OQueue_Cons].CurrPos, PcsVel:=zeroPCS); // PCS belt follow set up
	END_IF
END_IF

// stop management
outHalt(axesgroup := robot_group, Execute := state > 0 AND (NOT execute OR state = 15)
	, Deceleration:=RobotAccel * 10, Jerk:=RobotAccel * 10, BufferMode:=mcAborting
	,done => outHaltDone, error => outHaltErr);
OutStop(AxesGroup := robot_group, Execute := (NOT execute AND outHaltDone)
	, Deceleration:=RobotAccel * 10, Jerk:=RobotAccel * 10, BufferMode:=mcAborting
		, Done => outStopDone, error => outStopErr);

IF (state > 2 AND State <= 80) AND NOT execute THEN
		State:=80;
END_IF

//error check
IF (CameraError) THEN
	State:=101;
END_IF
IF (PowError) THEN
	State:=102;
END_IF	
IF ConnectionError THEN
	State:=100;
END_IF

CASE err103state OF
	0:
		err103_counter := 0;
		IF WrongWaitCycle THEN
			camerEnb := FALSE;
			err103state := 10;
		END_IF
	10:
		err103_timer(in:= TRUE, pt := T#5S);
		IF err103_timer.Q THEN
			err103state := 20;
		END_IF
	20:
		camerEnb := TRUE;
		err103_timer(in:= FALSE);
		err103state := 30;
	30:
		err103_timer(in:= TRUE, pt := T#2S);
		IF err103_timer.Q THEN
			IF WrongWaitCycle THEN
				State:=103;
				err103state := 40;
			ELSE
				err103state := err103_counter := 0;
			END_IF
		END_IF
	40:
		IF state = 0 THEN
			err103state := 0;
		END_IF
END_CASE

IF state > 80 THEN
	ready := waitting_for_obj := ready_to_pick := FALSE;
	error := TRUE;
END_IF

IF (NOT Enable) THEN
	State:=0;
END_IF

CASE State OF
//INIT
0:
	OQueue_Cons:=0;
	error
	:= ready
	:= waitting_for_obj
	:= ready_to_pick
	:= debugLook
	:= camerEnb
	:= FALSE;
	
	IF Enable THEN
		State:=1;
	END_IF

//power on axis
1:
	IF (PowReady) THEN
		camerEnb := TRUE;
		State:=2;
	END_IF

//WAIT for "execute"
2:
	ready := TRUE;
	waitting_for_obj := ready_to_pick := FALSE;
	GrMoveFb0(AxesGroup:=robot_group, Execute:=FALSE);
	GrMoveFb0_Lin(AxesGroup:=robot_group, Execute:=FALSE);
	IF (execute) THEN
		State:=10;
	END_IF

//Prepare for execution
10:
	GrMoveFb0(axesgroup := robot_group, execute := TRUE, position := ADR(safe_pos), coordsystem := mcacs
	, BufferMode:=mcAborting, TransitionMode:= tmNone, TransitionParameter:= ADR(GrRelCorner) 
	, OverFeedPerc:= safepoint_overfeed, Done=>GrMoveDone);
	IF GrMoveDone THEN
		State:=20;
	ELSIF (NOT execute) THEN
		State:=80;
	END_IF
		
// stop movement and go waitting
15:
	GrMoveFb0_Lin(AxesGroup:=robot_group, Execute:=FALSE);
	IF outStopDone THEN
		state := 20;
	END_IF
	
//move robot over ink deposit
20: 
	GrMoveFb0_Lin(AxesGroup:=robot_group, Execute:=TRUE, CoordSystem:=mcMcs, BufferMode:=buff_mod, 
			TransitionParameter:=ADR(GrRelCorner), Position:=ADR(WaittingUp), Velocity:=RobotSpeed, 
			Acceleration:=RobotAccel, Deceleration:=RobotAccel, Jerk:=RobotAccel*3, Done=>GrMoveDone);
				
	debugLook := TRUE;	// start photo
	
	// when done go on
	IF (GrMoveDone OR OQueue_Prod <> OQueue_Cons) AND NOT debugButton_2 THEN
		State:=30;
	ELSIF (NOT execute) THEN
		State:=80;
	END_IF

//prepare for group movement
30:
	GrMoveFb1(AxesGroup:=robot_group, Execute:=FALSE);
	GrMoveFb2(AxesGroup:=robot_group, Execute:=FALSE);
	GrMoveFb3(AxesGroup:=robot_group, Execute:=FALSE);
	GrMoveFb4(AxesGroup:=robot_group, Execute:=FALSE);
	GrMoveFb5(AxesGroup:=robot_group, Execute:=FALSE);
	GrMoveFb6(AxesGroup:=robot_group, Execute:=FALSE);
	GrMoveFb7(AxesGroup:=robot_group, Execute:=FALSE);
	GrMoveFb8(AxesGroup:=robot_group, Execute:=FALSE);
	
	IF (NOT execute) THEN
		State:=80;
	END_IF

	// Create PCS coordinates of product
	ObjPosDown[3]:=Z;
	ObjPosUp[3]:=Z+RobotZDelta;
	
	// check if there are objects
	IF (OQueue_Prod <> OQueue_Cons) AND NOT debugButton_3 THEN
		pos:=OQueue[OQueue_Cons].CurrPos[1];
		IF (pos < y_entry_bound) AND (pos > y_exit_bound) THEN
			State:=40;
			GrMoveFb0(AxesGroup:=robot_group, Execute:=FALSE);
			GrMoveFb0_Lin(AxesGroup:=robot_group, Execute:=FALSE);
			PickTimer(in:=FALSE);
		ELSE
			State:=20;
		END_IF

		// consume objects that are out of reachable area
		IF(pos<y_exit_bound) THEN
			OQueue_Cons := OQueue_Cons +1;
			IF OQueue_Cons>=32 THEN
				OQueue_Cons:=0;
			END_IF
		END_IF
	ELSIF state <> 80 AND NOT debugButton_3 THEN
		debugLook := FALSE;	// stop photo to clean all obj data for next pick cycle
		OQueue_Cons := 0;
		State:=20;
	ELSIF debugButton_3 AND debugButton_4 THEN
		State:=40;
	END_IF
	
//GROUP MOVEMENT
40:
	GrMoveFb3(AxesGroup:=robot_group, Execute:=TRUE, CoordSystem:=mcPcs, BufferMode:=buff_mod, TransitionMode:=tmRelativeCornerDistance, 
			TransitionParameter:=ADR(GrRelCorner), Position:=ADR(ObjPosUp), Velocity:=RobotSpeed, 
			Acceleration:=RobotAccel, Deceleration:=RobotAccel, Jerk:=RobotAccel*20);
	GrMoveFb4(AxesGroup:=robot_group, Execute:=TRUE, CoordSystem:=mcPcs, BufferMode:=buff_mod, TransitionMode:=tmRelativeCornerDistance, 
			TransitionParameter:=ADR(GrRelCorner), Position:=ADR(ObjPosDown), Velocity:=RobotSpeed, 
			Acceleration:=RobotAccel, Deceleration:=RobotAccel, Jerk:=RobotAccel*20, Done=>GrMoveDone);
	
	// when completed go on
	IF GrMoveDone THEN
		ready_to_pick := TRUE;
		PickTimer(in:=TRUE,pt:= delayTime);
		IF wait_signal_before_pick AND isPicked THEN
			IF PickTimer.Q THEN
				state := 41;
			END_IF
		ELSIF NOT wait_signal_before_pick THEN
			IF PickTimer.Q THEN
				state := 41;
			END_IF
		END_IF
	END_IF

	pos:=OQueue[OQueue_Cons].CurrPos[1];
	// consume objects that are out of reachable area
	IF(pos<y_exit_bound) AND NOT debugButton_3 THEN
		State := 15;
	END_IF
41:
	ready_to_pick := FALSE;
	PickTimer(in:=FALSE);
	State:=50;
	
//move back
50:
	GrMoveFb5(AxesGroup:=robot_group, Execute:=TRUE, CoordSystem:=mcPcs, BufferMode:=buff_mod, TransitionMode:=tmRelativeCornerDistance, 
			TransitionParameter:=ADR(GrRelCorner), Position:=ADR(ObjPosUp), Velocity:=RobotSpeed, 
			Acceleration:=RobotAccel, Deceleration:=RobotAccel, Jerk:=RobotAccel*10, Done=>GrMoveDone2);
			
	GrMoveFb6(AxesGroup:=robot_group, Execute:=TRUE, CoordSystem:=mcMcs, BufferMode:=buff_mod, TransitionMode:=tmRelativeCornerDistance, 
			TransitionParameter:=ADR(GrRelCorner), Position:=ADR(MarkerUp), Velocity:=RobotSpeed, 
			Acceleration:=RobotAccel, Deceleration:=RobotAccel, Jerk:=RobotAccel*10);

	GrMoveFb7(AxesGroup:=robot_group, Execute:=TRUE, CoordSystem:=mcMcs, BufferMode:=buff_mod, TransitionMode:=tmRelativeCornerDistance, 
			TransitionParameter:=ADR(GrRelCorner), Position:=ADR(MarkerDown), Velocity:=RobotSpeed, 
			Acceleration:=RobotAccel, Deceleration:=RobotAccel, Jerk:=RobotAccel*10, Done=>GrMoveDone2);

	// When completed, go on
	IF GrMoveDone2 THEN
		ready_to_release := TRUE;
		PickTimer(in := TRUE, pt := delay_release_obj);
		IF PickTimer.Q THEN
			ready_to_release := FALSE;
			PickTimer(in := FALSE);
			state:= 55;
		END_IF
	END_IF
	
55:
//*)
	GrMoveFb8(AxesGroup:=robot_group, Execute:=TRUE, CoordSystem:=mcMcs, BufferMode:=buff_mod, TransitionMode:=tmRelativeCornerDistance, 
			TransitionParameter:=ADR(GrRelCorner), Position:=ADR(MarkerUp), Velocity:=RobotSpeed, 
			Acceleration:=RobotAccel, Deceleration:=RobotAccel, Jerk:=RobotAccel*10, Done=>GrMoveDone3);
	// When completed, go on
	IF GrMoveDone3 THEN
		OQueue[OQueue_Cons].Id := 0;
		OQueue_Cons := OQueue_Cons +1;
		IF OQueue_Cons>=32 THEN
			OQueue_Cons:=0;
		END_IF
		State:= 30;
		Ev:=16#00;
	END_IF

//Stop the belt
80: 
	State:=2;

//ERROR states
100: //error on Client activation
101: //error on Camera activation
102: //error on axis power on
103: //number of waiting PLC cycles for Client Read-Write too small
END_CASE


// Feedback about next object position (DEBUG)
IF (OQueue_Prod<>OQueue_Cons) THEN
	NextObjPos:=OQueue[OQueue_Cons].CurrPos[2];
	NextObjPosX:=OQueue[OQueue_Cons].CurrPos[1];
	CameraObjN:=OQueue_Prod-OQueue_Cons;
	IF (CameraObjN<0) THEN
		CameraObjN:=CameraObjN-32;
	END_IF
ELSE
	NextObjPos:=0.0;
	NextObjPosX:=0.0;
	CameraObjN:=0;
END_IF

END_FUNCTION_BLOCK

// Device/Application/hand blocks/Grab_Control
FUNCTION_BLOCK Grab_Control
VAR_INPUT
	Enable : BOOL;
	OverFeed : INT;
	Grab : Grab_Command;
END_VAR
VAR_OUTPUT
	Done : BOOL;
	isMoving : BOOL;
	Error : BOOL;
	Err_Message : Error_Message;
END_VAR
VAR
	state : INT := 0;
	i : INT;
	//movment settings
	Finger_Movement: ArcaLibrary.MCAT_MoveDirectAbsolute;
	
	ReadCurrentPos : ArcaLibrary.MC_GroupReadActualPosition;
	CurrPos : ARRAY [1..6] OF REAL;
	CoordSys1: ArcaLibrary.MC_COORD_SYSTEM := mcMCS;
	
	Set1: ArcaLibrary.MCAT_Settings;
	ToolMoveVel:REAL:=100;
	ToolMoveAcc:REAL:=500;
	ToolMoveJrk:REAL:=2500;
	bufmode: ArcaLibrary.MC_BUFFER_MODE:=mcBuffered;
	transition: ArcaLibrary.MC_TRANSITION_MODE:=tmRelativeCornerDistance;
	tmPar: ARRAY [1..12] OF REAL :=[1.0, 1.0, 1.0, 1.0, 1.0, 1.0, 1.0, 1.0, 1.0, 1.0, 1.0, 1.0];

	Pos_For_Hand_Block : ArcaLibrary.MCAT_Position;
	Position_0: ARRAY [1..6] OF REAL :=[0.300, -0.100, 0.200, 160.0, 180.0, 0.0];
	Position_1: ARRAY [1..6] OF REAL :=[0.500, -0.100, 0.200, 160.0, 180.0, 0.0];
	RobotMovPos: ARRAY [1..6] OF REAL :=[0.50, -0.100, 0.200, 160.0, 180.0, 0.0];
	
	AxesPosForExternal: ARRAY [1..32] OF REAL;
	
	MaxDifference : REAL := 0.005;
	
	// grab pos
	g_grab: ARRAY [1..32] OF REAL;
	
	// max degree for every motor
	Root_min : REAL := 235;
	Root_max : REAL := 350;
	
	Tip_min : REAL := 140;
	Tip_max : REAL := 40;
	
	
	grab_angle_min : REAL := 0;
	grab_angle_max : REAL := 180;
	
	// debug
	mid_0_max: REAL;
	mid_0_min: REAL;
	
	clamp : Value_Clamp;
END_VAR

IF NOT Enable AND state > 0 THEN
	state := 0;
END_IF

IF overfeed > 90 THEN
	overfeed := 90;
ELSIF overfeed < 0 THEN
	overfeed := 0;
END_IF

// read current virtual robot postion
ReadCurrentPos(axesGroup := 0, execute := state > 0, CoordSystem:=mcMcs, Position=>CurrPos);
IF ReadCurrentPos.Error THEN
	state := -10;
END_IF

CASE state OF
	-30:
		error := TRUE;
		Err_Message := error_message.Err_AuxAxis_Movement_Block_err;
	-10:
	(*
		IF ReadCurrentPos.ErrorID THEN
			
		END_IF
	*)
		error := TRUE;
		Err_Message := error_message.Err_AuxAxis_Movement_Cannot_read_virture_robot_position;
		
	0:
		Done := error := FALSE;
		Err_Message := error_message.Err_None;
		
		IF Enable THEN
			state := 10;
		END_IF

	10:	//initialize
	
		// set position
		// clamp Root_Angle
		clamp(current := Grab.Root_Angle, first_value := Root_min, second_value := Root_max, newV => g_grab[1]);
		
		// clamp Tip_Angle
		clamp(current := Grab.Tip_Angle, first_value := Tip_min, second_value := Tip_max, newV => g_grab[2]);
		
		// clamp Tip_Angle
		clamp(current := Grab.Clamp_Angle, first_value := grab_angle_min, second_value := grab_angle_max, newV => g_grab[3]);
		
		// take a judge to find where is the robot and give a different destination
		IF ABS(CurrPos[1] - Position_0[1]) > MaxDifference THEN
			RobotMovPos := Position_0;
		ELSE 
			RobotMovPos := Position_1;
		END_IF
		
		// asign value for hand movment block
		Pos_For_Hand_Block.Position := RobotMovPos;
		Pos_For_Hand_Block.AxesPosition:=AxesPosForExternal;
		Pos_For_Hand_Block.AuxAxes:=g_grab;
		Pos_For_Hand_Block.CoordSystem:=CoordSys1;
		
		Set1.Velocity:=ToolMoveVel;
		Set1.Acceleration:=ToolMoveAcc;
		Set1.Deceleration:=ToolMoveAcc;
		Set1.Jerk:=ToolMoveJrk;
		Set1.OverfeedPerc:=Overfeed;
		Set1.BufferMode:=bufmode;
		Set1.TransitionMode:=transition;
		Set1.TransitionParameter:=tmPar;
		
		Finger_Movement(AxesGroup:=0, Execute:=FALSE);
		State := 20;
	20:
		IF (NOT enable) THEN
			State := 0;
		END_IF
		
		Finger_Movement(AxesGroup:=0, Execute:=TRUE, Position:=Pos_For_Hand_Block, Settings:=Set1, active => isMoving);
		
		IF Finger_Movement.Done THEN
			Finger_Movement(AxesGroup:=0, Execute:=FALSE);
			state := 50;
		ELSIF Finger_Movement.Error OR Finger_Movement.CommandAborted THEN
			state := -30;
		END_IF
	50:
		done := TRUE;
END_CASE
// end of the program

END_FUNCTION_BLOCK

// Device/Application/simple_functions/Value_Clamp
FUNCTION_BLOCK Value_Clamp
// clamp the input value between first value and second value
VAR_INPUT
	Current : REAL;
	First_Value : REAL;
	Second_value : REAL;
END_VAR
VAR_OUTPUT
	newV : REAL;
END_VAR
VAR
END_VAR

newV := Current;
IF First_Value < Second_value THEN
	IF Current < First_Value THEN
		newV := First_Value;
	END_IF
	IF Current > Second_value THEN
		newV := Second_value;
	END_IF
ELSIF First_Value > Second_value THEN
	IF Current > First_Value THEN
		newV := First_Value;
	END_IF
	IF Current < Second_value THEN
		newV := Second_value;
	END_IF
END_IF
// not going to deal the situation of first value equal to second value

END_FUNCTION_BLOCK

// Device/Application/hand blocks/Grab_Demo
FUNCTION_BLOCK Grab_Demo
VAR_INPUT
	enable :BOOL;
	internal_hand_enable : BOOL;
	startMov :BOOL;
	ovr : INT;
END_VAR

VAR_OUTPUT
	IsEnabled : BOOL;
	IsMoving : BOOL;
	err : BOOL;
	err_message : error_message;
END_VAR

VAR
	// state control
	cycleState : INT;	// state machine
	cycleCounter : INT;	// counte how many time already been done
	start_cycle : INT := 1;	// start cycle from a number
	total_cycle_time : INT := 24; //	max cycle time
	cycleTimer : ton;
	cycleDelayTime : TIME := T#500MS;	// delay time between every gesture
	
	// hand powerOn
	powerHand : BOOL;
	powerOnHand : AuxAxis_PowerOn;
	_enabled : BOOL;
	
	// gestrure mov block
	GrabMov : Grab_Control;
	GrabCmd : grab_command;
	_GrabCmdEmpt : grab_command;
END_VAR


//err
IF powerOnHand.Error OR GrabMov.Error THEN
	err := TRUE;
	IF powerOnHand.Error THEN
		err_message := powerOnHand.Err_Message;
	ELSIF GrabMov.Error THEN
		err_message := GrabMov.Err_Message;
	END_IF
ELSE
	err := FALSE;
	err_message := error_message.Err_None;
END_IF

// enable hand
IF internal_hand_enable THEN
	powerOnHand(enable := enable);
	_enabled := IsEnabled := powerOnHand.Done;
END_IF

IF NOT enable THEN
	cycleState := 0;
	isMoving := FALSE;
	cycleTimer(in := FALSE);	// reset timer
	GrabMov(Enable := FALSE);	// reset movement block
END_IF

CASE cycleState OF
	0: 
		// if block is enabled and order to move and (manager by internal power or by external power)
		IF enable AND startMov AND (NOT internal_hand_enable OR _enabled) THEN
			GrabCmd.Root_Angle := 200;	// all open
			GrabCmd.Tip_Angle := 200;
			GrabCmd.Clamp_Angle := 0;
			
			cycleCounter := start_cycle;	// set counter to start_cycle
			cycleState := 10;
		END_IF
	10:
		GrabMov(Enable := TRUE, overfeed := ovr,Grab := GrabCmd, isMoving => isMoving);
		IF GrabMov.Done THEN
			cycleTimer(in := TRUE, pt:= cycleDelayTime);	// start timer for delay
			IF cycleTimer.Q THEN	// time reach
				cycleCounter := cycleCounter + 1;	// done and self add for next gesture
				cycleTimer(in := FALSE);	// reset timer
				GrabMov(Enable := FALSE);	// reset movement block
				
				IF cycleCounter <= total_cycle_time THEN
					IF cycleCounter <= 5 THEN	// first movement, root as clamp
						IF GrabCmd.Root_Angle <> 400 THEN // if not clamp
							GrabCmd.Root_Angle := 400;	// root in max
							GrabCmd.Tip_Angle := 90;	// tip mov in middle
						ELSE
							GrabCmd.Root_Angle := 200;	// root in open
							GrabCmd.Tip_Angle := 200;	// tip in open
						END_IF
					ELSIF cycleCounter <= 9 THEN	// second movement, show tip movement
						IF GrabCmd.Tip_Angle <> 40 THEN // if not clmap
							GrabCmd.Root_Angle := 200;	// root in open
							GrabCmd.Tip_Angle := 40;	// tip max
						ELSE
							GrabCmd.Root_Angle := 200;	// root in open
							GrabCmd.Tip_Angle := 200;	// tip in open
						END_IF
					ELSIF cyclecounter <= 15 THEN	// second movement, tip as clamp
						IF GrabCmd.Tip_Angle <> 40 THEN
							GrabCmd.Root_Angle := 300;	// root mov to mid
							GrabCmd.Tip_Angle := 40;	// tip max
						ELSE
							GrabCmd.Root_Angle := 200;	// root in open
							GrabCmd.Tip_Angle := 140;	// tip in open
						END_IF
					ELSIF cyclecounter <= 18 THEN	// third movement, show clamp angle
						IF GrabCmd.Clamp_Angle <> 180 THEN
							GrabCmd.Clamp_Angle := 180;	// clamp angle to max
						ELSE
							GrabCmd.Clamp_Angle := 0;	// clamp angle to min
						END_IF
					ELSIF cyclecounter <= 24 THEN	// fouth movement, tip as clamp in another clamp angle
						IF GrabCmd.Tip_Angle <> 40 THEN
							GrabCmd.Root_Angle := 300;	// root mov to mid
							GrabCmd.Tip_Angle := 40;	// tip max
						ELSE
							GrabCmd.Root_Angle := 200;	// root in open
							GrabCmd.Tip_Angle := 140;	// tip in open
						END_IF
					END_IF
					cycleState := 10;	// if not reach total number then go back keep do next gesture
				ELSE
					cycleState := 0;	// if reach maximum then go back beginning
				END_IF
			END_IF
		END_IF
END_CASE

END_FUNCTION_BLOCK
